LIN {X 0,Y 363.671,Z 845.185,A -85,B 0,C 180,E1 12162.19,E2 12162.19} C_VEL
LIN {X 0,Y 361.588,Z 841.697,A -85,B 0,C 180,E1 12164.164,E2 12164.164} C_VEL
LIN {X 0,Y 357.251,Z 835.619,A -85,B 0,C 180,E1 12167.101,E2 12167.101} C_VEL
LIN {X 0,Y 357.31,Z 834.842,A -85,B 0,C 180,E1 12167.431,E2 12167.431} C_VEL
LIN {X 0,Y 361.071,Z 816.803,A -85,B 0,C 180,E1 12173.615,E2 12173.615} C_VEL
LIN {X 0,Y 366.874,Z 793.95,A -85,B 0,C 180,E1 12179.237,E2 12179.237} C_VEL
LIN {X 0,Y 375.007,Z 763.75,A -85,B 0,C 180,E1 12184.589,E2 12184.589} C_VEL
LIN {X 0,Y 383.635,Z 730.788,A -85,B 0,C 180,E1 12188.762,E2 12188.762} C_VEL
LIN {X 0,Y 391.479,Z 697.041,A -85,B 0,C 180,E1 12191.86,E2 12191.86} C_VEL
LIN {X 0,Y 398.91,Z 656.609,A -85,B 0,C 180,E1 12194.4,E2 12194.4} C_VEL
LIN {X 0,Y 399.383,Z 648.133,A -85,B 0,C 180,E1 12194.901,E2 12194.901} C_VEL
LIN {X 0,Y 385.814,Z 616.735,A -85,B 0,C 180,E1 12198.747,E2 12198.747} C_VEL
LIN {X 0,Y 368.99,Z 587.739,A -85,B 0,C 180,E1 12202.995,E2 12202.995} C_VEL
LIN {X 0,Y 356.259,Z 569.433,A -85,B 0,C 180,E1 12206.425,E2 12206.425} C_VEL
LIN {X 0,Y 353.406,Z 564.379,A -85,B 0,C 180,E1 12207.307,E2 12207.307} C_VEL
LIN {X 0,Y 353.308,Z 563.28,A -85,B 0,C 180,E1 12207.531,E2 12207.531} C_VEL
LIN {X 0,Y 353.587,Z 563.28,A -85,B 0,C 180,E1 12214.74,E2 12214.74} C_VEL
LIN {X 0,Y 353.926,Z 563.28,A -85,B 0,C 180,E1 12222.638,E2 12222.638} C_VEL
LIN {X 0,Y 354.275,Z 563.28,A -85,B 0,C 180,E1 12230.193,E2 12230.193} C_VEL
LIN {X 0,Y 354.927,Z 563.28,A -85,B 0,C 180,E1 12237.566,E2 12237.566} C_VEL
LIN {X 0,Y 354.696,Z 563.28,A -85,B 0,C 180,E1 12244.884,E2 12244.884} C_VEL
LIN {X 0,Y 354.337,Z 563.28,A -85,B 0,C 180,E1 12252.297,E2 12252.297} C_VEL
LIN {X 0,Y 353.84,Z 563.28,A -85,B 0,C 180,E1 12260.247,E2 12260.247} C_VEL
LIN {X 0,Y 353.553,Z 563.28,A -85,B 0,C 180,E1 12268.004,E2 12268.004} C_VEL
LIN {X 0,Y 353.436,Z 563.28,A -85,B 0,C 180,E1 12275.787,E2 12275.787} C_VEL
LIN {X 0,Y 353.192,Z 563.28,A -85,B 0,C 180,E1 12283.423,E2 12283.423} C_VEL
LIN {X 0,Y 353.306,Z 563.28,A -85,B 0,C 180,E1 12290.249,E2 12290.249} C_VEL
LIN {X 0,Y 353.41,Z 564.08,A -85,B 0,C 180,E1 12293.675,E2 12293.675} C_VEL
LIN {X 0,Y 355.308,Z 568.353,A -85,B 0,C 180,E1 12296.796,E2 12296.796} C_VEL
LIN {X 0,Y 359.309,Z 570.875,A -85,B 0,C 180,E1 12303.148,E2 12303.148} C_VEL
LIN {X 0,Y 360.621,Z 572.122,A -85,B 0,C 180,E1 12305.652,E2 12305.652} C_VEL
LIN {X 0,Y 362.642,Z 576.09,A -85,B 0,C 180,E1 12310.557,E2 12310.557} C_VEL
LIN {X 0,Y 364.977,Z 577.856,A -85,B 0,C 180,E1 12317.261,E2 12317.261} C_VEL
LIN {X 0,Y 366.337,Z 578.371,A -85,B 0,C 180,E1 12322.903,E2 12322.903} C_VEL
LIN {X 0,Y 366.937,Z 578.462,A -85,B 0,C 180,E1 12330.001,E2 12330.001} C_VEL
LIN {X 0,Y 366.335,Z 578.387,A -85,B 0,C 180,E1 12337.1,E2 12337.1} C_VEL
LIN {X 0,Y 364.743,Z 577.75,A -85,B 0,C 180,E1 12343.57,E2 12343.57} C_VEL
LIN {X 0,Y 362.374,Z 575.801,A -85,B 0,C 180,E1 12350.065,E2 12350.065} C_VEL
LIN {X 0,Y 360.594,Z 571.886,A -85,B 0,C 180,E1 12354.449,E2 12354.449} C_VEL
LIN {X 0,Y 356.588,Z 569.679,A -85,B 0,C 180,E1 12361.221,E2 12361.221} C_VEL
LIN {X 0,Y 353.659,Z 565.515,A -85,B 0,C 180,E1 12365.832,E2 12365.832} C_VEL
LIN {X 0,Y 353.31,Z 563.28,A -85,B 0,C 180,E1 12366.725,E2 12366.725} C_VEL
LIN {X 0,Y 353.255,Z 563.28,A -85,B 0,C 180,E1 12373.429,E2 12373.429} C_VEL
LIN {X 0,Y 353.304,Z 563.28,A -85,B 0,C 180,E1 12380.248,E2 12380.248} C_VEL
LIN {X 0,Y 353.291,Z 563.28,A -85,B 0,C 180,E1 12386.268,E2 12386.268} C_VEL
LIN {X 0,Y 353.514,Z 563.28,A -85,B 0,C 180,E1 12393.692,E2 12393.692} C_VEL
LIN {X 0,Y 353.865,Z 563.28,A -85,B 0,C 180,E1 12400.051,E2 12400.051} C_VEL
LIN {X 0,Y 354.167,Z 563.28,A -85,B 0,C 180,E1 12407.697,E2 12407.697} C_VEL
LIN {X 0,Y 354.686,Z 563.28,A -85,B 0,C 180,E1 12415.116,E2 12415.116} C_VEL
LIN {X 0,Y 354.947,Z 563.28,A -85,B 0,C 180,E1 12419.997,E2 12419.997} C_VEL
LIN {X 0,Y 354.533,Z 563.28,A -85,B 0,C 180,E1 12427.333,E2 12427.333} C_VEL
LIN {X 0,Y 354.204,Z 563.28,A -85,B 0,C 180,E1 12434.807,E2 12434.807} C_VEL
LIN {X 0,Y 353.755,Z 563.28,A -85,B 0,C 180,E1 12442.573,E2 12442.573} C_VEL
LIN {X 0,Y 353.544,Z 563.28,A -85,B 0,C 180,E1 12447.999,E2 12447.999} C_VEL
LIN {X 0,Y 353.5,Z 563.901,A -85,B 0,C 180,E1 12452.699,E2 12452.699} C_VEL
LIN {X 0,Y 356.151,Z 569.235,A -85,B 0,C 180,E1 12453.542,E2 12453.542} C_VEL
LIN {X 0,Y 358.926,Z 573.181,A -85,B 0,C 180,E1 12454.336,E2 12454.336} C_VEL
LIN {X 0,Y 373.428,Z 594.714,A -85,B 0,C 180,E1 12458.126,E2 12458.126} C_VEL
LIN {X 0,Y 389.979,Z 625.192,A -85,B 0,C 180,E1 12462.337,E2 12462.337} C_VEL
LIN {X 0,Y 399.94,Z 650.173,A -85,B 0,C 180,E1 12465.308,E2 12465.308} C_VEL
LIN {X 0,Y 393.844,Z 685.837,A -85,B 0,C 180,E1 12467.335,E2 12467.335} C_VEL
LIN {X 0,Y 385.413,Z 723.656,A -85,B 0,C 180,E1 12470.49,E2 12470.49} C_VEL
LIN {X 0,Y 377.04,Z 756.232,A -85,B 0,C 180,E1 12474.349,E2 12474.349} C_VEL
LIN {X 0,Y 368.957,Z 786.062,A -85,B 0,C 180,E1 12479.185,E2 12479.185} C_VEL
LIN {X 0,Y 362.194,Z 812.082,A -85,B 0,C 180,E1 12485.048,E2 12485.048} C_VEL
LIN {X 0,Y 358.052,Z 830.361,A -85,B 0,C 180,E1 12490.811,E2 12490.811} C_VEL
LIN {X 0,Y 355.896,Z 844.415,A -85,B 0,C 180,E1 12497.199,E2 12497.199} C_VEL
LIN {X 0,Y 355.194,Z 851.737,A -85,B 0,C 180,E1 12502.676,E2 12502.676} C_VEL
LIN {X 0,Y 355.069,Z 854.938,A -85,B 0,C 180,E1 12507.563,E2 12507.563} C_VEL
LIN {X 0,Y 355.088,Z 854.939,A -85,B 0,C 180,E1 12512.434,E2 12512.434} C_VEL
LIN {X 0,Y 355.305,Z 850.4,A -85,B 0,C 180,E1 12518.547,E2 12518.547} C_VEL
LIN {X 0,Y 356.324,Z 840.794,A -85,B 0,C 180,E1 12524.719,E2 12524.719} C_VEL
LIN {X 0,Y 357.31,Z 834.842,A -85,B 0,C 180,E1 12527.431,E2 12527.431} C_VEL
LIN {X 0,Y 356.685,Z 831.732,A -85,B 0,C 180,E1 12528.738,E2 12528.738} C_VEL
LIN {X 0,Y 352.209,Z 822.528,A -85,B 0,C 180,E1 12532.298,E2 12532.298} C_VEL
LIN {X 0,Y 352.36,Z 821.58,A -85,B 0,C 180,E1 12532.62,E2 12532.62} C_VEL
LIN {X 0,Y 358.152,Z 799.224,A -85,B 0,C 180,E1 12538.636,E2 12538.636} C_VEL
LIN {X 0,Y 365.443,Z 773.594,A -85,B 0,C 180,E1 12543.697,E2 12543.697} C_VEL
LIN {X 0,Y 374.852,Z 740.263,A -85,B 0,C 180,E1 12548.426,E2 12548.426} C_VEL
LIN {X 0,Y 383.311,Z 706.501,A -85,B 0,C 180,E1 12551.853,E2 12551.853} C_VEL
LIN {X 0,Y 391.215,Z 668.882,A -85,B 0,C 180,E1 12554.532,E2 12554.532} C_VEL
LIN {X 0,Y 393.652,Z 652,A -85,B 0,C 180,E1 12555.466,E2 12555.466} C_VEL
LIN {X 0,Y 380.35,Z 620.223,A -85,B 0,C 180,E1 12559.517,E2 12559.517} C_VEL
LIN {X 0,Y 364.483,Z 592.576,A -85,B 0,C 180,E1 12563.775,E2 12563.775} C_VEL
LIN {X 0,Y 351.882,Z 574.587,A -85,B 0,C 180,E1 12567.315,E2 12567.315} C_VEL
LIN {X 0,Y 348.505,Z 569.513,A -85,B 0,C 180,E1 12568.377,E2 12568.377} C_VEL
LIN {X 0,Y 345.524,Z 564.479,A -85,B 0,C 180,E1 12569.381,E2 12569.381} C_VEL
LIN {X 0,Y 345.407,Z 563.28,A -85,B 0,C 180,E1 12569.696,E2 12569.696} C_VEL
LIN {X 0,Y 345.745,Z 563.28,A -85,B 0,C 180,E1 12576.874,E2 12576.874} C_VEL
LIN {X 0,Y 346.098,Z 563.28,A -85,B 0,C 180,E1 12584.838,E2 12584.838} C_VEL
LIN {X 0,Y 346.567,Z 563.28,A -85,B 0,C 180,E1 12592.497,E2 12592.497} C_VEL
LIN {X 0,Y 347.065,Z 563.28,A -85,B 0,C 180,E1 12600.003,E2 12600.003} C_VEL
LIN {X 0,Y 346.585,Z 563.28,A -85,B 0,C 180,E1 12607.508,E2 12607.508} C_VEL
LIN {X 0,Y 346.201,Z 563.28,A -85,B 0,C 180,E1 12615.163,E2 12615.163} C_VEL
LIN {X 0,Y 345.783,Z 563.28,A -85,B 0,C 180,E1 12623.129,E2 12623.129} C_VEL
LIN {X 0,Y 345.532,Z 563.28,A -85,B 0,C 180,E1 12629.142,E2 12629.142} C_VEL
LIN {X 0,Y 345.496,Z 563.28,A -85,B 0,C 180,E1 12634.599,E2 12634.599} C_VEL
LIN {X 0,Y 345.221,Z 563.28,A -85,B 0,C 180,E1 12642.006,E2 12642.006} C_VEL
LIN {X 0,Y 345.236,Z 564.112,A -85,B 0,C 180,E1 12644.299,E2 12644.299} C_VEL
LIN {X 0,Y 347.221,Z 568.468,A -85,B 0,C 180,E1 12647.012,E2 12647.012} C_VEL
LIN {X 0,Y 352.224,Z 571.904,A -85,B 0,C 180,E1 12653.411,E2 12653.411} C_VEL
LIN {X 0,Y 354.534,Z 576.458,A -85,B 0,C 180,E1 12657.128,E2 12657.128} C_VEL
LIN {X 0,Y 358.695,Z 578.802,A -85,B 0,C 180,E1 12663.756,E2 12663.756} C_VEL
LIN {X 0,Y 359.613,Z 580.385,A -85,B 0,C 180,E1 12665.675,E2 12665.675} C_VEL
LIN {X 0,Y 362.06,Z 584.381,A -85,B 0,C 180,E1 12671.471,E2 12671.471} C_VEL
LIN {X 0,Y 364.301,Z 585.783,A -85,B 0,C 180,E1 12678.048,E2 12678.048} C_VEL
LIN {X 0,Y 365.704,Z 586.297,A -85,B 0,C 180,E1 12685.267,E2 12685.267} C_VEL
LIN {X 0,Y 365.909,Z 586.287,A -85,B 0,C 180,E1 12692.365,E2 12692.365} C_VEL
LIN {X 0,Y 364.899,Z 586.104,A -85,B 0,C 180,E1 12699.523,E2 12699.523} C_VEL
LIN {X 0,Y 362.809,Z 584.931,A -85,B 0,C 180,E1 12706.621,E2 12706.621} C_VEL
LIN {X 0,Y 360.101,Z 581.658,A -85,B 0,C 180,E1 12713.228,E2 12713.228} C_VEL
LIN {X 0,Y 359.173,Z 578.883,A -85,B 0,C 180,E1 12715.463,E2 12715.463} C_VEL
LIN {X 0,Y 354.995,Z 577.053,A -85,B 0,C 180,E1 12722.14,E2 12722.14} C_VEL
LIN {X 0,Y 352.286,Z 572.512,A -85,B 0,C 180,E1 12726.42,E2 12726.42} C_VEL
LIN {X 0,Y 351.69,Z 571.028,A -85,B 0,C 180,E1 12727.405,E2 12727.405} C_VEL
LIN {X 0,Y 347.021,Z 568.132,A -85,B 0,C 180,E1 12733.255,E2 12733.255} C_VEL
LIN {X 0,Y 345.297,Z 564.151,A -85,B 0,C 180,E1 12735.632,E2 12735.632} C_VEL
LIN {X 0,Y 345.257,Z 563.28,A -85,B 0,C 180,E1 12737.991,E2 12737.991} C_VEL
LIN {X 0,Y 345.341,Z 563.28,A -85,B 0,C 180,E1 12745.383,E2 12745.383} C_VEL
LIN {X 0,Y 345.466,Z 563.28,A -85,B 0,C 180,E1 12751.28,E2 12751.28} C_VEL
LIN {X 0,Y 345.767,Z 563.28,A -85,B 0,C 180,E1 12756.87,E2 12756.87} C_VEL
LIN {X 0,Y 346.086,Z 563.28,A -85,B 0,C 180,E1 12764.832,E2 12764.832} C_VEL
LIN {X 0,Y 346.582,Z 563.28,A -85,B 0,C 180,E1 12772.492,E2 12772.492} C_VEL
LIN {X 0,Y 347.047,Z 563.28,A -85,B 0,C 180,E1 12777.505,E2 12777.505} C_VEL
LIN {X 0,Y 346.768,Z 563.28,A -85,B 0,C 180,E1 12784.99,E2 12784.99} C_VEL
LIN {X 0,Y 346.396,Z 563.28,A -85,B 0,C 180,E1 12792.578,E2 12792.578} C_VEL
LIN {X 0,Y 345.901,Z 563.28,A -85,B 0,C 180,E1 12800.423,E2 12800.423} C_VEL
LIN {X 0,Y 345.693,Z 563.28,A -85,B 0,C 180,E1 12805.878,E2 12805.878} C_VEL
LIN {X 0,Y 345.599,Z 564.041,A -85,B 0,C 180,E1 12810.622,E2 12810.622} C_VEL
LIN {X 0,Y 348.222,Z 569.222,A -85,B 0,C 180,E1 12811.537,E2 12811.537} C_VEL
LIN {X 0,Y 350.847,Z 572.607,A -85,B 0,C 180,E1 12812.349,E2 12812.349} C_VEL
LIN {X 0,Y 366.964,Z 596.388,A -85,B 0,C 180,E1 12816.899,E2 12816.899} C_VEL
LIN {X 0,Y 383.207,Z 626.372,A -85,B 0,C 180,E1 12821.302,E2 12821.302} C_VEL
LIN {X 0,Y 393.715,Z 651.973,A -85,B 0,C 180,E1 12824.541,E2 12824.541} C_VEL
LIN {X 0,Y 387.168,Z 689.313,A -85,B 0,C 180,E1 12826.802,E2 12826.802} C_VEL
LIN {X 0,Y 378.838,Z 724.988,A -85,B 0,C 180,E1 12829.868,E2 12829.868} C_VEL
LIN {X 0,Y 369.612,Z 759.114,A -85,B 0,C 180,E1 12834.062,E2 12834.062} C_VEL
LIN {X 0,Y 361.647,Z 786.824,A -85,B 0,C 180,E1 12838.727,E2 12838.727} C_VEL
LIN {X 0,Y 355.017,Z 810.994,A -85,B 0,C 180,E1 12844.275,E2 12844.275} C_VEL
LIN {X 0,Y 350.395,Z 830.074,A -85,B 0,C 180,E1 12850.361,E2 12850.361} C_VEL
LIN {X 0,Y 348.045,Z 844.165,A -85,B 0,C 180,E1 12856.906,E2 12856.906} C_VEL
LIN {X 0,Y 347.317,Z 851.491,A -85,B 0,C 180,E1 12862.509,E2 12862.509} C_VEL
LIN {X 0,Y 347.117,Z 854.922,A -85,B 0,C 180,E1 12868.878,E2 12868.878} C_VEL
LIN {X 0,Y 347.209,Z 854.695,A -85,B 0,C 180,E1 12872.49,E2 12872.49} C_VEL
LIN {X 0,Y 347.42,Z 850.153,A -85,B 0,C 180,E1 12878.743,E2 12878.743} C_VEL
LIN {X 0,Y 348.528,Z 840.543,A -85,B 0,C 180,E1 12885.056,E2 12885.056} C_VEL
LIN {X 0,Y 351.495,Z 825.207,A -85,B 0,C 180,E1 12891.401,E2 12891.401} C_VEL
LIN {X 0,Y 352.36,Z 821.58,A -85,B 0,C 180,E1 12892.62,E2 12892.62} C_VEL
LIN {X 0,Y 350.509,Z 813.946,A -85,B 0,C 180,E1 12895.176,E2 12895.176} C_VEL
LIN {X 0,Y 349.082,Z 805.529,A -85,B 0,C 180,E1 12897.691,E2 12897.691} C_VEL
LIN {X 0,Y 356.46,Z 780.665,A -85,B 0,C 180,E1 12903.09,E2 12903.09} C_VEL
LIN {X 0,Y 365.494,Z 750.497,A -85,B 0,C 180,E1 12907.888,E2 12907.888} C_VEL
LIN {X 0,Y 374.925,Z 716.168,A -85,B 0,C 180,E1 12911.766,E2 12911.766} C_VEL
LIN {X 0,Y 382.897,Z 681.994,A -85,B 0,C 180,E1 12914.525,E2 12914.525} C_VEL
LIN {X 0,Y 387.365,Z 654.079,A -85,B 0,C 180,E1 12916.257,E2 12916.257} C_VEL
LIN {X 0,Y 374.283,Z 622.504,A -85,B 0,C 180,E1 12920.489,E2 12920.489} C_VEL
LIN {X 0,Y 358.211,Z 594.506,A -85,B 0,C 180,E1 12925.078,E2 12925.078} C_VEL
LIN {X 0,Y 345.012,Z 575.716,A -85,B 0,C 180,E1 12929.078,E2 12929.078} C_VEL
LIN {X 0,Y 340.974,Z 569.777,A -85,B 0,C 180,E1 12930.466,E2 12930.466} C_VEL
LIN {X 0,Y 337.71,Z 564.923,A -85,B 0,C 180,E1 12931.661,E2 12931.661} C_VEL
LIN {X 0,Y 337.55,Z 563.28,A -85,B 0,C 180,E1 12932.01,E2 12932.01} C_VEL
LIN {X 0,Y 337.978,Z 563.28,A -85,B 0,C 180,E1 12939.651,E2 12939.651} C_VEL
LIN {X 0,Y 338.288,Z 563.28,A -85,B 0,C 180,E1 12947.116,E2 12947.116} C_VEL
LIN {X 0,Y 338.825,Z 563.28,A -85,B 0,C 180,E1 12954.892,E2 12954.892} C_VEL
LIN {X 0,Y 339.163,Z 563.28,A -85,B 0,C 180,E1 12960.003,E2 12960.003} C_VEL
LIN {X 0,Y 338.65,Z 563.28,A -85,B 0,C 180,E1 12967.685,E2 12967.685} C_VEL
LIN {X 0,Y 338.26,Z 563.28,A -85,B 0,C 180,E1 12975.528,E2 12975.528} C_VEL
LIN {X 0,Y 337.94,Z 563.28,A -85,B 0,C 180,E1 12980.932,E2 12980.932} C_VEL
LIN {X 0,Y 337.687,Z 563.28,A -85,B 0,C 180,E1 12986.657,E2 12986.657} C_VEL
LIN {X 0,Y 337.582,Z 563.28,A -85,B 0,C 180,E1 12992.442,E2 12992.442} C_VEL
LIN {X 0,Y 337.414,Z 564.037,A -85,B 0,C 180,E1 12996.425,E2 12996.425} C_VEL
LIN {X 0,Y 339.634,Z 568.903,A -85,B 0,C 180,E1 12999.18,E2 12999.18} C_VEL
LIN {X 0,Y 343.94,Z 571.904,A -85,B 0,C 180,E1 13003.953,E2 13003.953} C_VEL
LIN {X 0,Y 346.648,Z 576.829,A -85,B 0,C 180,E1 13007.56,E2 13007.56} C_VEL
LIN {X 0,Y 351.098,Z 579.793,A -85,B 0,C 180,E1 13013.224,E2 13013.224} C_VEL
LIN {X 0,Y 353.773,Z 584.552,A -85,B 0,C 180,E1 13017.461,E2 13017.461} C_VEL
LIN {X 0,Y 357.821,Z 586.644,A -85,B 0,C 180,E1 13023.906,E2 13023.906} C_VEL
LIN {X 0,Y 358.684,Z 588.701,A -85,B 0,C 180,E1 13025.848,E2 13025.848} C_VEL
LIN {X 0,Y 361.176,Z 592.319,A -85,B 0,C 180,E1 13031.74,E2 13031.74} C_VEL
LIN {X 0,Y 363.326,Z 593.607,A -85,B 0,C 180,E1 13038.016,E2 13038.016} C_VEL
LIN {X 0,Y 364.74,Z 594.137,A -85,B 0,C 180,E1 13045.255,E2 13045.255} C_VEL
LIN {X 0,Y 364.949,Z 594.099,A -85,B 0,C 180,E1 13052.371,E2 13052.371} C_VEL
LIN {X 0,Y 363.929,Z 593.942,A -85,B 0,C 180,E1 13059.548,E2 13059.548} C_VEL
LIN {X 0,Y 361.909,Z 592.826,A -85,B 0,C 180,E1 13066.457,E2 13066.457} C_VEL
LIN {X 0,Y 359.176,Z 589.635,A -85,B 0,C 180,E1 13073.105,E2 13073.105} C_VEL
LIN {X 0,Y 358.173,Z 586.719,A -85,B 0,C 180,E1 13075.539,E2 13075.539} C_VEL
LIN {X 0,Y 354.029,Z 584.918,A -85,B 0,C 180,E1 13082.137,E2 13082.137} C_VEL
LIN {X 0,Y 351.143,Z 580.278,A -85,B 0,C 180,E1 13086.644,E2 13086.644} C_VEL
LIN {X 0,Y 350.271,Z 578.746,A -85,B 0,C 180,E1 13087.99,E2 13087.99} C_VEL
LIN {X 0,Y 345.694,Z 575.627,A -85,B 0,C 180,E1 13093.655,E2 13093.655} C_VEL
LIN {X 0,Y 343.38,Z 570.929,A -85,B 0,C 180,E1 13096.755,E2 13096.755} C_VEL
LIN {X 0,Y 338.699,Z 567.666,A -85,B 0,C 180,E1 13101.883,E2 13101.883} C_VEL
LIN {X 0,Y 337.303,Z 563.589,A -85,B 0,C 180,E1 13103.736,E2 13103.736} C_VEL
LIN {X 0,Y 337.518,Z 563.28,A -85,B 0,C 180,E1 13110.539,E2 13110.539} C_VEL
LIN {X 0,Y 337.832,Z 563.28,A -85,B 0,C 180,E1 13116.294,E2 13116.294} C_VEL
LIN {X 0,Y 338.024,Z 563.28,A -85,B 0,C 180,E1 13121.788,E2 13121.788} C_VEL
LIN {X 0,Y 338.409,Z 563.28,A -85,B 0,C 180,E1 13129.723,E2 13129.723} C_VEL
LIN {X 0,Y 339.128,Z 563.28,A -85,B 0,C 180,E1 13137.447,E2 13137.447} C_VEL
LIN {X 0,Y 338.842,Z 563.28,A -85,B 0,C 180,E1 13145.107,E2 13145.107} C_VEL
LIN {X 0,Y 338.468,Z 563.28,A -85,B 0,C 180,E1 13152.877,E2 13152.877} C_VEL
LIN {X 0,Y 337.924,Z 563.28,A -85,B 0,C 180,E1 13160.928,E2 13160.928} C_VEL
LIN {X 0,Y 337.632,Z 563.573,A -85,B 0,C 180,E1 13168.256,E2 13168.256} C_VEL
LIN {X 0,Y 339.813,Z 568.738,A -85,B 0,C 180,E1 13169.146,E2 13169.146} C_VEL
LIN {X 0,Y 342.794,Z 572.041,A -85,B 0,C 180,E1 13170.154,E2 13170.154} C_VEL
LIN {X 0,Y 359.439,Z 596.205,A -85,B 0,C 180,E1 13175.279,E2 13175.279} C_VEL
LIN {X 0,Y 376.137,Z 626.656,A -85,B 0,C 180,E1 13180.099,E2 13180.099} C_VEL
LIN {X 0,Y 387.721,Z 655.219,A -85,B 0,C 180,E1 13183.885,E2 13183.885} C_VEL
LIN {X 0,Y 380.122,Z 694.653,A -85,B 0,C 180,E1 13186.388,E2 13186.388} C_VEL
LIN {X 0,Y 371.641,Z 728.551,A -85,B 0,C 180,E1 13189.482,E2 13189.482} C_VEL
LIN {X 0,Y 362.163,Z 761.995,A -85,B 0,C 180,E1 13193.76,E2 13193.76} C_VEL
LIN {X 0,Y 353.372,Z 790.825,A -85,B 0,C 180,E1 13198.916,E2 13198.916} C_VEL
LIN {X 0,Y 346.823,Z 813.809,A -85,B 0,C 180,E1 13204.553,E2 13204.553} C_VEL
LIN {X 0,Y 342.012,Z 833.157,A -85,B 0,C 180,E1 13211.226,E2 13211.226} C_VEL
LIN {X 0,Y 340.079,Z 845.195,A -85,B 0,C 180,E1 13217.456,E2 13217.456} C_VEL
LIN {X 0,Y 339.298,Z 852.286,A -85,B 0,C 180,E1 13223.615,E2 13223.615} C_VEL
LIN {X 0,Y 339.347,Z 854.854,A -85,B 0,C 180,E1 13229.999,E2 13229.999} C_VEL
LIN {X 0,Y 339.254,Z 853.243,A -85,B 0,C 180,E1 13235.103,E2 13235.103} C_VEL
LIN {X 0,Y 339.811,Z 846.898,A -85,B 0,C 180,E1 13241.387,E2 13241.387} C_VEL
LIN {X 0,Y 341.78,Z 834.894,A -85,B 0,C 180,E1 13248.001,E2 13248.001} C_VEL
LIN {X 0,Y 345.864,Z 817.46,A -85,B 0,C 180,E1 13254.348,E2 13254.348} C_VEL
LIN {X 0,Y 349.082,Z 805.529,A -85,B 0,C 180,E1 13257.691,E2 13257.691} C_VEL
LIN {X 0,Y 348.158,Z 796.543,A -85,B 0,C 180,E1 13260.162,E2 13260.162} C_VEL
LIN {X 0,Y 347.612,Z 786.819,A -85,B 0,C 180,E1 13262.567,E2 13262.567} C_VEL
LIN {X 0,Y 356.551,Z 758.624,A -85,B 0,C 180,E1 13267.471,E2 13267.471} C_VEL
LIN {X 0,Y 366.415,Z 725.473,A -85,B 0,C 180,E1 13271.648,E2 13271.648} C_VEL
LIN {X 0,Y 375.662,Z 688.407,A -85,B 0,C 180,E1 13274.914,E2 13274.914} C_VEL
LIN {X 0,Y 381.562,Z 657.868,A -85,B 0,C 180,E1 13276.843,E2 13276.843} C_VEL
LIN {X 0,Y 368.955,Z 626.366,A -85,B 0,C 180,E1 13281.241,E2 13281.241} C_VEL
LIN {X 0,Y 353.883,Z 599.562,A -85,B 0,C 180,E1 13285.859,E2 13285.859} C_VEL
LIN {X 0,Y 338.477,Z 576.893,A -85,B 0,C 180,E1 13290.911,E2 13290.911} C_VEL
LIN {X 0,Y 333.198,Z 569.859,A -85,B 0,C 180,E1 13292.892,E2 13292.892} C_VEL
LIN {X 0,Y 329.909,Z 564.995,A -85,B 0,C 180,E1 13294.255,E2 13294.255} C_VEL
LIN {X 0,Y 329.721,Z 563.28,A -85,B 0,C 180,E1 13294.601,E2 13294.601} C_VEL
LIN {X 0,Y 330.058,Z 563.28,A -85,B 0,C 180,E1 13301.338,E2 13301.338} C_VEL
LIN {X 0,Y 330.487,Z 563.28,A -85,B 0,C 180,E1 13309.479,E2 13309.479} C_VEL
LIN {X 0,Y 331.192,Z 563.28,A -85,B 0,C 180,E1 13317.391,E2 13317.391} C_VEL
LIN {X 0,Y 331.128,Z 563.28,A -85,B 0,C 180,E1 13322.615,E2 13322.615} C_VEL
LIN {X 0,Y 330.585,Z 563.28,A -85,B 0,C 180,E1 13330.523,E2 13330.523} C_VEL
LIN {X 0,Y 330.139,Z 563.28,A -85,B 0,C 180,E1 13338.663,E2 13338.663} C_VEL
LIN {X 0,Y 329.844,Z 563.28,A -85,B 0,C 180,E1 13344.317,E2 13344.317} C_VEL
LIN {X 0,Y 329.741,Z 563.921,A -85,B 0,C 180,E1 13349.428,E2 13349.428} C_VEL
LIN {X 0,Y 331.188,Z 567.963,A -85,B 0,C 180,E1 13351.118,E2 13351.118} C_VEL
LIN {X 0,Y 336.08,Z 571.903,A -85,B 0,C 180,E1 13356.081,E2 13356.081} C_VEL
LIN {X 0,Y 339.131,Z 577.222,A -85,B 0,C 180,E1 13359.702,E2 13359.702} C_VEL
LIN {X 0,Y 342.728,Z 579.756,A -85,B 0,C 180,E1 13363.696,E2 13363.696} C_VEL
LIN {X 0,Y 345.917,Z 584.941,A -85,B 0,C 180,E1 13367.871,E2 13367.871} C_VEL
LIN {X 0,Y 349.963,Z 587.64,A -85,B 0,C 180,E1 13373.013,E2 13373.013} C_VEL
LIN {X 0,Y 352.937,Z 592.55,A -85,B 0,C 180,E1 13377.667,E2 13377.667} C_VEL
LIN {X 0,Y 356.873,Z 594.489,A -85,B 0,C 180,E1 13383.942,E2 13383.942} C_VEL
LIN {X 0,Y 359.25,Z 599.08,A -85,B 0,C 180,E1 13389.33,E2 13389.33} C_VEL
LIN {X 0,Y 361.583,Z 601.103,A -85,B 0,C 180,E1 13395.5,E2 13395.5} C_VEL
LIN {X 0,Y 362.967,Z 601.698,A -85,B 0,C 180,E1 13400.429,E2 13400.429} C_VEL
LIN {X 0,Y 363.979,Z 602.001,A -85,B 0,C 180,E1 13407.625,E2 13407.625} C_VEL
LIN {X 0,Y 363.777,Z 601.961,A -85,B 0,C 180,E1 13414.76,E2 13414.76} C_VEL
LIN {X 0,Y 362.345,Z 601.471,A -85,B 0,C 180,E1 13422.02,E2 13422.02} C_VEL
LIN {X 0,Y 360.067,Z 599.989,A -85,B 0,C 180,E1 13428.754,E2 13428.754} C_VEL
LIN {X 0,Y 357.467,Z 595.699,A -85,B 0,C 180,E1 13434.797,E2 13434.797} C_VEL
LIN {X 0,Y 356.218,Z 594.331,A -85,B 0,C 180,E1 13437.173,E2 13437.173} C_VEL
LIN {X 0,Y 352.058,Z 591.704,A -85,B 0,C 180,E1 13443.697,E2 13443.697} C_VEL
LIN {X 0,Y 349.743,Z 586.894,A -85,B 0,C 180,E1 13447.393,E2 13447.393} C_VEL
LIN {X 0,Y 344.721,Z 583.586,A -85,B 0,C 180,E1 13453.639,E2 13453.639} C_VEL
LIN {X 0,Y 342.364,Z 578.741,A -85,B 0,C 180,E1 13456.807,E2 13456.807} C_VEL
LIN {X 0,Y 337.545,Z 575.41,A -85,B 0,C 180,E1 13462.067,E2 13462.067} C_VEL
LIN {X 0,Y 335.829,Z 571.039,A -85,B 0,C 180,E1 13464.255,E2 13464.255} C_VEL
LIN {X 0,Y 331.03,Z 567.877,A -85,B 0,C 180,E1 13469.032,E2 13469.032} C_VEL
LIN {X 0,Y 329.64,Z 563.879,A -85,B 0,C 180,E1 13470.65,E2 13470.65} C_VEL
LIN {X 0,Y 329.953,Z 563.28,A -85,B 0,C 180,E1 13478.536,E2 13478.536} C_VEL
LIN {X 0,Y 330.323,Z 563.28,A -85,B 0,C 180,E1 13486.794,E2 13486.794} C_VEL
LIN {X 0,Y 330.922,Z 563.28,A -85,B 0,C 180,E1 13494.765,E2 13494.765} C_VEL
LIN {X 0,Y 331.237,Z 563.28,A -85,B 0,C 180,E1 13499.997,E2 13499.997} C_VEL
LIN {X 0,Y 330.732,Z 563.28,A -85,B 0,C 180,E1 13507.864,E2 13507.864} C_VEL
LIN {X 0,Y 330.308,Z 563.28,A -85,B 0,C 180,E1 13515.906,E2 13515.906} C_VEL
LIN {X 0,Y 329.831,Z 563.28,A -85,B 0,C 180,E1 13524.312,E2 13524.312} C_VEL
LIN {X 0,Y 329.753,Z 563.28,A -85,B 0,C 180,E1 13525.583,E2 13525.583} C_VEL
LIN {X 0,Y 331.649,Z 568.354,A -85,B 0,C 180,E1 13526.514,E2 13526.514} C_VEL
LIN {X 0,Y 335.135,Z 572.196,A -85,B 0,C 180,E1 13527.846,E2 13527.846} C_VEL
LIN {X 0,Y 348.91,Z 591.676,A -85,B 0,C 180,E1 13532.577,E2 13532.577} C_VEL
LIN {X 0,Y 363.161,Z 615.427,A -85,B 0,C 180,E1 13536.984,E2 13536.984} C_VEL
LIN {X 0,Y 376.647,Z 644.281,A -85,B 0,C 180,E1 13541.335,E2 13541.335} C_VEL
LIN {X 0,Y 381.733,Z 658.528,A -85,B 0,C 180,E1 13543.238,E2 13543.238} C_VEL
LIN {X 0,Y 373.746,Z 697.132,A -85,B 0,C 180,E1 13545.746,E2 13545.746} C_VEL
LIN {X 0,Y 364.397,Z 732.195,A -85,B 0,C 180,E1 13549.093,E2 13549.093} C_VEL
LIN {X 0,Y 355.331,Z 762.729,A -85,B 0,C 180,E1 13553.139,E2 13553.139} C_VEL
LIN {X 0,Y 346.061,Z 791.659,A -85,B 0,C 180,E1 13558.447,E2 13558.447} C_VEL
LIN {X 0,Y 339.141,Z 814.626,A -85,B 0,C 180,E1 13564.288,E2 13564.288} C_VEL
LIN {X 0,Y 334.271,Z 833.191,A -85,B 0,C 180,E1 13570.894,E2 13570.894} C_VEL
LIN {X 0,Y 332.178,Z 845.347,A -85,B 0,C 180,E1 13577.434,E2 13577.434} C_VEL
LIN {X 0,Y 331.421,Z 852.04,A -85,B 0,C 180,E1 13583.463,E2 13583.463} C_VEL
LIN {X 0,Y 331.46,Z 854.609,A -85,B 0,C 180,E1 13589.999,E2 13589.999} C_VEL
LIN {X 0,Y 331.383,Z 852.041,A -85,B 0,C 180,E1 13596.536,E2 13596.536} C_VEL
LIN {X 0,Y 332.265,Z 844.545,A -85,B 0,C 180,E1 13603.124,E2 13603.124} C_VEL
LIN {X 0,Y 334.73,Z 831.569,A -85,B 0,C 180,E1 13609.759,E2 13609.759} C_VEL
LIN {X 0,Y 339.744,Z 812.489,A -85,B 0,C 180,E1 13616.368,E2 13616.368} C_VEL
LIN {X 0,Y 347.424,Z 787.397,A -85,B 0,C 180,E1 13622.446,E2 13622.446} C_VEL
LIN {X 0,Y 347.612,Z 786.819,A -85,B 0,C 180,E1 13622.567,E2 13622.567} C_VEL
LIN {X 0,Y 347.5,Z 776.544,A -85,B 0,C 180,E1 13624.909,E2 13624.909} C_VEL
LIN {X 0,Y 347.789,Z 765.564,A -85,B 0,C 180,E1 13627.155,E2 13627.155} C_VEL
LIN {X 0,Y 357.563,Z 734.561,A -85,B 0,C 180,E1 13631.455,E2 13631.455} C_VEL
LIN {X 0,Y 367.487,Z 698.723,A -85,B 0,C 180,E1 13634.987,E2 13634.987} C_VEL
LIN {X 0,Y 375.599,Z 660.92,A -85,B 0,C 180,E1 13637.539,E2 13637.539} C_VEL
LIN {X 0,Y 363.254,Z 629.59,A -85,B 0,C 180,E1 13642.14,E2 13642.14} C_VEL
LIN {X 0,Y 348.592,Z 602.601,A -85,B 0,C 180,E1 13647.009,E2 13647.009} C_VEL
LIN {X 0,Y 334.877,Z 582.819,A -85,B 0,C 180,E1 13651.765,E2 13651.765} C_VEL
LIN {X 0,Y 330.133,Z 576.371,A -85,B 0,C 180,E1 13653.629,E2 13653.629} C_VEL
LIN {X 0,Y 326.103,Z 570.274,A -85,B 0,C 180,E1 13655.392,E2 13655.392} C_VEL
LIN {X 0,Y 322.21,Z 565.269,A -85,B 0,C 180,E1 13657.211,E2 13657.211} C_VEL
LIN {X 0,Y 321.969,Z 563.28,A -85,B 0,C 180,E1 13657.696,E2 13657.696} C_VEL
LIN {X 0,Y 322.235,Z 563.28,A -85,B 0,C 180,E1 13663.685,E2 13663.685} C_VEL
LIN {X 0,Y 322.747,Z 563.28,A -85,B 0,C 180,E1 13671.94,E2 13671.94} C_VEL
LIN {X 0,Y 323.271,Z 563.28,A -85,B 0,C 180,E1 13677.327,E2 13677.327} C_VEL
LIN {X 0,Y 323.211,Z 563.28,A -85,B 0,C 180,E1 13682.679,E2 13682.679} C_VEL
LIN {X 0,Y 322.65,Z 563.28,A -85,B 0,C 180,E1 13690.847,E2 13690.847} C_VEL
LIN {X 0,Y 322.337,Z 563.28,A -85,B 0,C 180,E1 13696.316,E2 13696.316} C_VEL
LIN {X 0,Y 322.038,Z 563.667,A -85,B 0,C 180,E1 13703.973,E2 13703.973} C_VEL
LIN {X 0,Y 323.67,Z 568.384,A -85,B 0,C 180,E1 13705.407,E2 13705.407} C_VEL
LIN {X 0,Y 328.207,Z 571.991,A -85,B 0,C 180,E1 13709.058,E2 13709.058} C_VEL
LIN {X 0,Y 331.249,Z 576.956,A -85,B 0,C 180,E1 13712.123,E2 13712.123} C_VEL
LIN {X 0,Y 334.857,Z 579.898,A -85,B 0,C 180,E1 13715.865,E2 13715.865} C_VEL
LIN {X 0,Y 338.432,Z 585.297,A -85,B 0,C 180,E1 13719.995,E2 13719.995} C_VEL
LIN {X 0,Y 341.539,Z 587.571,A -85,B 0,C 180,E1 13723.471,E2 13723.471} C_VEL
LIN {X 0,Y 345.072,Z 592.881,A -85,B 0,C 180,E1 13728.026,E2 13728.026} C_VEL
LIN {X 0,Y 348.838,Z 595.42,A -85,B 0,C 180,E1 13732.801,E2 13732.801} C_VEL
LIN {X 0,Y 351.974,Z 600.412,A -85,B 0,C 180,E1 13737.683,E2 13737.683} C_VEL
LIN {X 0,Y 356.292,Z 603.018,A -85,B 0,C 180,E1 13744.696,E2 13744.696} C_VEL
LIN {X 0,Y 358.582,Z 607.286,A -85,B 0,C 180,E1 13750.118,E2 13750.118} C_VEL
LIN {X 0,Y 360.929,Z 609.081,A -85,B 0,C 180,E1 13756.574,E2 13756.574} C_VEL
LIN {X 0,Y 362.475,Z 609.702,A -85,B 0,C 180,E1 13762.827,E2 13762.827} C_VEL
LIN {X 0,Y 363.089,Z 609.804,A -85,B 0,C 180,E1 13770.001,E2 13770.001} C_VEL
LIN {X 0,Y 362.469,Z 609.744,A -85,B 0,C 180,E1 13777.176,E2 13777.176} C_VEL
LIN {X 0,Y 360.814,Z 609.034,A -85,B 0,C 180,E1 13783.923,E2 13783.923} C_VEL
LIN {X 0,Y 358.266,Z 606.892,A -85,B 0,C 180,E1 13790.73,E2 13790.73} C_VEL
LIN {X 0,Y 355.931,Z 602.346,A -85,B 0,C 180,E1 13796.011,E2 13796.011} C_VEL
LIN {X 0,Y 351.705,Z 600.281,A -85,B 0,C 180,E1 13802.701,E2 13802.701} C_VEL
LIN {X 0,Y 348.776,Z 595.406,A -85,B 0,C 180,E1 13807.282,E2 13807.282} C_VEL
LIN {X 0,Y 343.444,Z 591.115,A -85,B 0,C 180,E1 13814.003,E2 13814.003} C_VEL
LIN {X 0,Y 341.015,Z 586.484,A -85,B 0,C 180,E1 13817.204,E2 13817.204} C_VEL
LIN {X 0,Y 336.294,Z 583.01,A -85,B 0,C 180,E1 13822.366,E2 13822.366} C_VEL
LIN {X 0,Y 333.983,Z 578.67,A -85,B 0,C 180,E1 13825.119,E2 13825.119} C_VEL
LIN {X 0,Y 329.242,Z 574.66,A -85,B 0,C 180,E1 13829.871,E2 13829.871} C_VEL
LIN {X 0,Y 327.44,Z 570.882,A -85,B 0,C 180,E1 13831.654,E2 13831.654} C_VEL
LIN {X 0,Y 322.948,Z 567.333,A -85,B 0,C 180,E1 13835.129,E2 13835.129} C_VEL
LIN {X 0,Y 322.039,Z 563.28,A -85,B 0,C 180,E1 13836.256,E2 13836.256} C_VEL
LIN {X 0,Y 322.239,Z 563.28,A -85,B 0,C 180,E1 13843.679,E2 13843.679} C_VEL
LIN {X 0,Y 322.761,Z 563.28,A -85,B 0,C 180,E1 13851.934,E2 13851.934} C_VEL
LIN {X 0,Y 323.287,Z 563.28,A -85,B 0,C 180,E1 13857.322,E2 13857.322} C_VEL
LIN {X 0,Y 323.179,Z 563.28,A -85,B 0,C 180,E1 13862.673,E2 13862.673} C_VEL
LIN {X 0,Y 322.665,Z 563.28,A -85,B 0,C 180,E1 13870.848,E2 13870.848} C_VEL
LIN {X 0,Y 322.35,Z 563.28,A -85,B 0,C 180,E1 13876.309,E2 13876.309} C_VEL
LIN {X 0,Y 321.99,Z 563.385,A -85,B 0,C 180,E1 13882.591,E2 13882.591} C_VEL
LIN {X 0,Y 323.8,Z 568.301,A -85,B 0,C 180,E1 13883.606,E2 13883.606} C_VEL
LIN {X 0,Y 327.325,Z 571.877,A -85,B 0,C 180,E1 13885.147,E2 13885.147} C_VEL
LIN {X 0,Y 333.711,Z 581.227,A -85,B 0,C 180,E1 13887.792,E2 13887.792} C_VEL
LIN {X 0,Y 343.182,Z 594.556,A -85,B 0,C 180,E1 13891.203,E2 13891.203} C_VEL
LIN {X 0,Y 357.42,Z 617.945,A -85,B 0,C 180,E1 13895.901,E2 13895.901} C_VEL
LIN {X 0,Y 370.95,Z 647.719,A -85,B 0,C 180,E1 13900.604,E2 13900.604} C_VEL
LIN {X 0,Y 375.597,Z 662.076,A -85,B 0,C 180,E1 13902.559,E2 13902.559} C_VEL
LIN {X 0,Y 367.564,Z 698.728,A -85,B 0,C 180,E1 13905.025,E2 13905.025} C_VEL
LIN {X 0,Y 357.593,Z 734.543,A -85,B 0,C 180,E1 13908.546,E2 13908.546} C_VEL
LIN {X 0,Y 347.628,Z 766.008,A -85,B 0,C 180,E1 13912.918,E2 13912.918} C_VEL
LIN {X 0,Y 338.183,Z 794.381,A -85,B 0,C 180,E1 13918.378,E2 13918.378} C_VEL
LIN {X 0,Y 330.481,Z 818.657,A -85,B 0,C 180,E1 13925.015,E2 13925.015} C_VEL
LIN {X 0,Y 326.262,Z 834.381,A -85,B 0,C 180,E1 13931.108,E2 13931.108} C_VEL
LIN {X 0,Y 324.217,Z 846.015,A -85,B 0,C 180,E1 13937.78,E2 13937.78} C_VEL
LIN {X 0,Y 323.479,Z 852.75,A -85,B 0,C 180,E1 13944.645,E2 13944.645} C_VEL
LIN {X 0,Y 323.561,Z 854.364,A -85,B 0,C 180,E1 13949.999,E2 13949.999} C_VEL
LIN {X 0,Y 323.511,Z 851.795,A -85,B 0,C 180,E1 13956.695,E2 13956.695} C_VEL
LIN {X 0,Y 324.459,Z 844.296,A -85,B 0,C 180,E1 13963.446,E2 13963.446} C_VEL
LIN {X 0,Y 327.066,Z 831.312,A -85,B 0,C 180,E1 13970.244,E2 13970.244} C_VEL
LIN {X 0,Y 332.425,Z 812.234,A -85,B 0,C 180,E1 13976.995,E2 13976.995} C_VEL
LIN {X 0,Y 340.444,Z 787.461,A -85,B 0,C 180,E1 13983.116,E2 13983.116} C_VEL
LIN {X 0,Y 347.789,Z 765.564,A -85,B 0,C 180,E1 13987.155,E2 13987.155} C_VEL
LIN {X 0,Y 348.437,Z 754.02,A -85,B 0,C 180,E1 13989.321,E2 13989.321} C_VEL
LIN {X 0,Y 349.154,Z 741.862,A -85,B 0,C 180,E1 13991.391,E2 13991.391} C_VEL
LIN {X 0,Y 359.251,Z 708.28,A -85,B 0,C 180,E1 13995.029,E2 13995.029} C_VEL
LIN {X 0,Y 368.775,Z 669.481,A -85,B 0,C 180,E1 13997.915,E2 13997.915} C_VEL
LIN {X 0,Y 369.36,Z 663.289,A -85,B 0,C 180,E1 13998.374,E2 13998.374} C_VEL
LIN {X 0,Y 357.97,Z 633.456,A -85,B 0,C 180,E1 14002.956,E2 14002.956} C_VEL
LIN {X 0,Y 344.724,Z 608.406,A -85,B 0,C 180,E1 14007.681,E2 14007.681} C_VEL
LIN {X 0,Y 331.226,Z 588.249,A -85,B 0,C 180,E1 14012.702,E2 14012.702} C_VEL
LIN {X 0,Y 323.205,Z 576.993,A -85,B 0,C 180,E1 14016.166,E2 14016.166} C_VEL
LIN {X 0,Y 319.553,Z 571.213,A -85,B 0,C 180,E1 14018.012,E2 14018.012} C_VEL
LIN {X 0,Y 314.646,Z 565.98,A -85,B 0,C 180,E1 14020.661,E2 14020.661} C_VEL
LIN {X 0,Y 314.171,Z 563.28,A -85,B 0,C 180,E1 14021.267,E2 14021.267} C_VEL
LIN {X 0,Y 314.591,Z 563.28,A -85,B 0,C 180,E1 14028.941,E2 14028.941} C_VEL
LIN {X 0,Y 315.365,Z 563.28,A -85,B 0,C 180,E1 14037.26,E2 14037.26} C_VEL
LIN {X 0,Y 315.316,Z 563.28,A -85,B 0,C 180,E1 14042.746,E2 14042.746} C_VEL
LIN {X 0,Y 314.741,Z 563.28,A -85,B 0,C 180,E1 14051.059,E2 14051.059} C_VEL
LIN {X 0,Y 314.261,Z 563.28,A -85,B 0,C 180,E1 14059.279,E2 14059.279} C_VEL
LIN {X 0,Y 316.144,Z 568.549,A -85,B 0,C 180,E1 14060.836,E2 14060.836} C_VEL
LIN {X 0,Y 320.382,Z 572.141,A -85,B 0,C 180,E1 14063.605,E2 14063.605} C_VEL
LIN {X 0,Y 323.431,Z 577.104,A -85,B 0,C 180,E1 14066.026,E2 14066.026} C_VEL
LIN {X 0,Y 326.782,Z 579.712,A -85,B 0,C 180,E1 14068.725,E2 14068.725} C_VEL
LIN {X 0,Y 330.263,Z 584.891,A -85,B 0,C 180,E1 14072.131,E2 14072.131} C_VEL
LIN {X 0,Y 333.641,Z 587.665,A -85,B 0,C 180,E1 14075.625,E2 14075.625} C_VEL
LIN {X 0,Y 337.232,Z 593.016,A -85,B 0,C 180,E1 14079.773,E2 14079.773} C_VEL
LIN {X 0,Y 340.321,Z 595.292,A -85,B 0,C 180,E1 14083.198,E2 14083.198} C_VEL
LIN {X 0,Y 344.094,Z 600.763,A -85,B 0,C 180,E1 14088.027,E2 14088.027} C_VEL
LIN {X 0,Y 347.758,Z 603.344,A -85,B 0,C 180,E1 14092.666,E2 14092.666} C_VEL
LIN {X 0,Y 351.141,Z 608.406,A -85,B 0,C 180,E1 14097.886,E2 14097.886} C_VEL
LIN {X 0,Y 355.301,Z 611.12,A -85,B 0,C 180,E1 14104.703,E2 14104.703} C_VEL
LIN {X 0,Y 357.961,Z 615.546,A -85,B 0,C 180,E1 14110.898,E2 14110.898} C_VEL
LIN {X 0,Y 360.4,Z 617.081,A -85,B 0,C 180,E1 14117.917,E2 14117.917} C_VEL
LIN {X 0,Y 361.847,Z 617.656,A -85,B 0,C 180,E1 14125.217,E2 14125.217} C_VEL
LIN {X 0,Y 362.06,Z 617.621,A -85,B 0,C 180,E1 14132.39,E2 14132.39} C_VEL
LIN {X 0,Y 361.013,Z 617.456,A -85,B 0,C 180,E1 14139.626,E2 14139.626} C_VEL
LIN {X 0,Y 358.954,Z 616.294,A -85,B 0,C 180,E1 14146.605,E2 14146.605} C_VEL
LIN {X 0,Y 356.14,Z 613.076,A -85,B 0,C 180,E1 14153.393,E2 14153.393} C_VEL
LIN {X 0,Y 354.581,Z 610.067,A -85,B 0,C 180,E1 14156.653,E2 14156.653} C_VEL
LIN {X 0,Y 350.386,Z 607.759,A -85,B 0,C 180,E1 14163.273,E2 14163.273} C_VEL
LIN {X 0,Y 347.508,Z 602.686,A -85,B 0,C 180,E1 14167.753,E2 14167.753} C_VEL
LIN {X 0,Y 342.321,Z 598.873,A -85,B 0,C 180,E1 14174.179,E2 14174.179} C_VEL
LIN {X 0,Y 339.51,Z 594.153,A -85,B 0,C 180,E1 14177.775,E2 14177.775} C_VEL
LIN {X 0,Y 334.926,Z 590.382,A -85,B 0,C 180,E1 14182.827,E2 14182.827} C_VEL
LIN {X 0,Y 332.867,Z 586.464,A -85,B 0,C 180,E1 14185.257,E2 14185.257} C_VEL
LIN {X 0,Y 327.963,Z 582.312,A -85,B 0,C 180,E1 14190.139,E2 14190.139} C_VEL
LIN {X 0,Y 325.9,Z 578.531,A -85,B 0,C 180,E1 14192.113,E2 14192.113} C_VEL
LIN {X 0,Y 321.277,Z 574.607,A -85,B 0,C 180,E1 14195.588,E2 14195.588} C_VEL
LIN {X 0,Y 319.364,Z 570.73,A -85,B 0,C 180,E1 14197.109,E2 14197.109} C_VEL
LIN {X 0,Y 314.984,Z 566.828,A -85,B 0,C 180,E1 14199.918,E2 14199.918} C_VEL
LIN {X 0,Y 314.189,Z 563.28,A -85,B 0,C 180,E1 14200.716,E2 14200.716} C_VEL
LIN {X 0,Y 314.606,Z 563.28,A -85,B 0,C 180,E1 14208.936,E2 14208.936} C_VEL
LIN {X 0,Y 315.381,Z 563.28,A -85,B 0,C 180,E1 14217.255,E2 14217.255} C_VEL
LIN {X 0,Y 315.291,Z 563.28,A -85,B 0,C 180,E1 14222.74,E2 14222.74} C_VEL
LIN {X 0,Y 314.757,Z 563.28,A -85,B 0,C 180,E1 14231.053,E2 14231.053} C_VEL
LIN {X 0,Y 314.273,Z 563.803,A -85,B 0,C 180,E1 14238.999,E2 14238.999} C_VEL
LIN {X 0,Y 316.389,Z 568.807,A -85,B 0,C 180,E1 14240.388,E2 14240.388} C_VEL
LIN {X 0,Y 319.702,Z 571.671,A -85,B 0,C 180,E1 14242.081,E2 14242.081} C_VEL
LIN {X 0,Y 324.099,Z 577.654,A -85,B 0,C 180,E1 14244.221,E2 14244.221} C_VEL
LIN {X 0,Y 338.892,Z 599.046,A -85,B 0,C 180,E1 14250.223,E2 14250.223} C_VEL
LIN {X 0,Y 353.328,Z 623.778,A -85,B 0,C 180,E1 14255.355,E2 14255.355} C_VEL
LIN {X 0,Y 365.964,Z 652.937,A -85,B 0,C 180,E1 14260.108,E2 14260.108} C_VEL
LIN {X 0,Y 369.596,Z 665.144,A -85,B 0,C 180,E1 14261.829,E2 14261.829} C_VEL
LIN {X 0,Y 361.031,Z 701.709,A -85,B 0,C 180,E1 14264.403,E2 14264.403} C_VEL
LIN {X 0,Y 350.807,Z 736.889,A -85,B 0,C 180,E1 14267.976,E2 14267.976} C_VEL
LIN {X 0,Y 339.96,Z 769.225,A -85,B 0,C 180,E1 14272.677,E2 14272.677} C_VEL
LIN {X 0,Y 330.547,Z 795.987,A -85,B 0,C 180,E1 14278.089,E2 14278.089} C_VEL
LIN {X 0,Y 322.773,Z 819.463,A -85,B 0,C 180,E1 14284.746,E2 14284.746} C_VEL
LIN {X 0,Y 318.21,Z 835.88,A -85,B 0,C 180,E1 14291.508,E2 14291.508} C_VEL
LIN {X 0,Y 316.355,Z 845.765,A -85,B 0,C 180,E1 14297.471,E2 14297.471} C_VEL
LIN {X 0,Y 315.596,Z 852.504,A -85,B 0,C 180,E1 14304.511,E2 14304.511} C_VEL
LIN {X 0,Y 315.672,Z 854.119,A -85,B 0,C 180,E1 14309.999,E2 14309.999} C_VEL
LIN {X 0,Y 315.623,Z 851.548,A -85,B 0,C 180,E1 14316.863,E2 14316.863} C_VEL
LIN {X 0,Y 316.617,Z 844.046,A -85,B 0,C 180,E1 14323.785,E2 14323.785} C_VEL
LIN {X 0,Y 319.441,Z 831.059,A -85,B 0,C 180,E1 14330.749,E2 14330.749} C_VEL
LIN {X 0,Y 325.171,Z 811.981,A -85,B 0,C 180,E1 14337.648,E2 14337.648} C_VEL
LIN {X 0,Y 333.829,Z 786.616,A -85,B 0,C 180,E1 14344.012,E2 14344.012} C_VEL
LIN {X 0,Y 343.565,Z 758.753,A -85,B 0,C 180,E1 14349.027,E2 14349.027} C_VEL
LIN {X 0,Y 349.154,Z 741.862,A -85,B 0,C 180,E1 14351.391,E2 14351.391} C_VEL
LIN {X 0,Y 350.158,Z 729.125,A -85,B 0,C 180,E1 14353.366,E2 14353.366} C_VEL
LIN {X 0,Y 350.838,Z 717.61,A -85,B 0,C 180,E1 14355.018,E2 14355.018} C_VEL
LIN {X 0,Y 351.319,Z 715.797,A -85,B 0,C 180,E1 14355.209,E2 14355.209} C_VEL
LIN {X 0,Y 360.563,Z 681.795,A -85,B 0,C 180,E1 14358.046,E2 14358.046} C_VEL
LIN {X 0,Y 363.516,Z 666.608,A -85,B 0,C 180,E1 14359.095,E2 14359.095} C_VEL
LIN {X 0,Y 353.113,Z 638.211,A -85,B 0,C 180,E1 14363.639,E2 14363.639} C_VEL
LIN {X 0,Y 340.693,Z 614.049,A -85,B 0,C 180,E1 14368.383,E2 14368.383} C_VEL
LIN {X 0,Y 328.698,Z 595.191,A -85,B 0,C 180,E1 14373.181,E2 14373.181} C_VEL
LIN {X 0,Y 320.555,Z 583.688,A -85,B 0,C 180,E1 14376.876,E2 14376.876} C_VEL
LIN {X 0,Y 316.1,Z 577.474,A -85,B 0,C 180,E1 14379.207,E2 14379.207} C_VEL
LIN {X 0,Y 312.367,Z 572.268,A -85,B 0,C 180,E1 14381.429,E2 14381.429} C_VEL
LIN {X 0,Y 310.671,Z 570.353,A -85,B 0,C 180,E1 14382.513,E2 14382.513} C_VEL
LIN {X 0,Y 306.742,Z 565.403,A -85,B 0,C 180,E1 14385.417,E2 14385.417} C_VEL
LIN {X 0,Y 306.543,Z 563.28,A -85,B 0,C 180,E1 14386.118,E2 14386.118} C_VEL
LIN {X 0,Y 307.12,Z 563.28,A -85,B 0,C 180,E1 14394.364,E2 14394.364} C_VEL
LIN {X 0,Y 307.57,Z 563.28,A -85,B 0,C 180,E1 14400.003,E2 14400.003} C_VEL
LIN {X 0,Y 306.929,Z 563.28,A -85,B 0,C 180,E1 14408.485,E2 14408.485} C_VEL
LIN {X 0,Y 306.592,Z 563.614,A -85,B 0,C 180,E1 14414.751,E2 14414.751} C_VEL
LIN {X 0,Y 308.388,Z 568.348,A -85,B 0,C 180,E1 14416.38,E2 14416.38} C_VEL
LIN {X 0,Y 312.43,Z 572.103,A -85,B 0,C 180,E1 14419.03,E2 14419.03} C_VEL
LIN {X 0,Y 316.113,Z 577.423,A -85,B 0,C 180,E1 14421.461,E2 14421.461} C_VEL
LIN {X 0,Y 318.728,Z 579.752,A -85,B 0,C 180,E1 14423.204,E2 14423.204} C_VEL
LIN {X 0,Y 322.234,Z 584.902,A -85,B 0,C 180,E1 14425.889,E2 14425.889} C_VEL
LIN {X 0,Y 325.486,Z 587.628,A -85,B 0,C 180,E1 14428.484,E2 14428.484} C_VEL
LIN {X 0,Y 329.694,Z 593.154,A -85,B 0,C 180,E1 14432.575,E2 14432.575} C_VEL
LIN {X 0,Y 332.444,Z 595.562,A -85,B 0,C 180,E1 14435.421,E2 14435.421} C_VEL
LIN {X 0,Y 336.199,Z 600.845,A -85,B 0,C 180,E1 14439.721,E2 14439.721} C_VEL
LIN {X 0,Y 339.205,Z 603.267,A -85,B 0,C 180,E1 14443.078,E2 14443.078} C_VEL
LIN {X 0,Y 343.387,Z 608.785,A -85,B 0,C 180,E1 14448.339,E2 14448.339} C_VEL
LIN {X 0,Y 346.691,Z 611.188,A -85,B 0,C 180,E1 14452.531,E2 14452.531} C_VEL
LIN {X 0,Y 350.045,Z 616.17,A -85,B 0,C 180,E1 14457.714,E2 14457.714} C_VEL
LIN {X 0,Y 354.252,Z 618.922,A -85,B 0,C 180,E1 14464.54,E2 14464.54} C_VEL
LIN {X 0,Y 356.864,Z 623.288,A -85,B 0,C 180,E1 14470.631,E2 14470.631} C_VEL
LIN {X 0,Y 359.019,Z 624.745,A -85,B 0,C 180,E1 14476.634,E2 14476.634} C_VEL
LIN {X 0,Y 360.545,Z 625.339,A -85,B 0,C 180,E1 14482.788,E2 14482.788} C_VEL
LIN {X 0,Y 361.163,Z 625.485,A -85,B 0,C 180,E1 14490.001,E2 14490.001} C_VEL
LIN {X 0,Y 360.539,Z 625.381,A -85,B 0,C 180,E1 14497.214,E2 14497.214} C_VEL
LIN {X 0,Y 358.875,Z 624.685,A -85,B 0,C 180,E1 14504,E2 14504} C_VEL
LIN {X 0,Y 356.297,Z 622.55,A -85,B 0,C 180,E1 14510.85,E2 14510.85} C_VEL
LIN {X 0,Y 353.763,Z 617.944,A -85,B 0,C 180,E1 14516.388,E2 14516.388} C_VEL
LIN {X 0,Y 349.621,Z 615.858,A -85,B 0,C 180,E1 14522.921,E2 14522.921} C_VEL
LIN {X 0,Y 346.45,Z 610.773,A -85,B 0,C 180,E1 14527.81,E2 14527.81} C_VEL
LIN {X 0,Y 341.112,Z 606.472,A -85,B 0,C 180,E1 14534.481,E2 14534.481} C_VEL
LIN {X 0,Y 338.332,Z 601.919,A -85,B 0,C 180,E1 14538.006,E2 14538.006} C_VEL
LIN {X 0,Y 333.64,Z 597.967,A -85,B 0,C 180,E1 14543.139,E2 14543.139} C_VEL
LIN {X 0,Y 331.256,Z 594.077,A -85,B 0,C 180,E1 14545.881,E2 14545.881} C_VEL
LIN {X 0,Y 326.372,Z 589.559,A -85,B 0,C 180,E1 14550.625,E2 14550.625} C_VEL
LIN {X 0,Y 324.305,Z 586.167,A -85,B 0,C 180,E1 14552.542,E2 14552.542} C_VEL
LIN {X 0,Y 319.606,Z 581.784,A -85,B 0,C 180,E1 14556.087,E2 14556.087} C_VEL
LIN {X 0,Y 317.461,Z 578.224,A -85,B 0,C 180,E1 14557.647,E2 14557.647} C_VEL
LIN {X 0,Y 312.984,Z 573.649,A -85,B 0,C 180,E1 14560.548,E2 14560.548} C_VEL
LIN {X 0,Y 311.4,Z 570.676,A -85,B 0,C 180,E1 14561.637,E2 14561.637} C_VEL
LIN {X 0,Y 306.845,Z 565.867,A -85,B 0,C 180,E1 14564.866,E2 14564.866} C_VEL
LIN {X 0,Y 306.446,Z 563.28,A -85,B 0,C 180,E1 14565.468,E2 14565.468} C_VEL
LIN {X 0,Y 306.945,Z 563.28,A -85,B 0,C 180,E1 14573.195,E2 14573.195} C_VEL
LIN {X 0,Y 307.539,Z 563.28,A -85,B 0,C 180,E1 14579.997,E2 14579.997} C_VEL
LIN {X 0,Y 306.942,Z 563.28,A -85,B 0,C 180,E1 14588.478,E2 14588.478} C_VEL
LIN {X 0,Y 306.658,Z 563.86,A -85,B 0,C 180,E1 14594.384,E2 14594.384} C_VEL
LIN {X 0,Y 308.582,Z 568.538,A -85,B 0,C 180,E1 14596.081,E2 14596.081} C_VEL
LIN {X 0,Y 312.271,Z 571.791,A -85,B 0,C 180,E1 14598.486,E2 14598.486} C_VEL
LIN {X 0,Y 315.942,Z 577.383,A -85,B 0,C 180,E1 14600.713,E2 14600.713} C_VEL
LIN {X 0,Y 318.197,Z 580.365,A -85,B 0,C 180,E1 14601.926,E2 14601.926} C_VEL
LIN {X 0,Y 327.51,Z 593.105,A -85,B 0,C 180,E1 14606.303,E2 14606.303} C_VEL
LIN {X 0,Y 341.358,Z 614.882,A -85,B 0,C 180,E1 14611.849,E2 14611.849} C_VEL
LIN {X 0,Y 353.796,Z 639.995,A -85,B 0,C 180,E1 14616.661,E2 14616.661} C_VEL
LIN {X 0,Y 363.502,Z 666.563,A -85,B 0,C 180,E1 14620.898,E2 14620.898} C_VEL
LIN {X 0,Y 354.756,Z 703.888,A -85,B 0,C 180,E1 14623.686,E2 14623.686} C_VEL
LIN {X 0,Y 344.436,Z 737.855,A -85,B 0,C 180,E1 14627.227,E2 14627.227} C_VEL
LIN {X 0,Y 332.979,Z 770.522,A -85,B 0,C 180,E1 14632.095,E2 14632.095} C_VEL
LIN {X 0,Y 323.194,Z 796.913,A -85,B 0,C 180,E1 14637.618,E2 14637.618} C_VEL
LIN {X 0,Y 315.418,Z 819.21,A -85,B 0,C 180,E1 14644.114,E2 14644.114} C_VEL
LIN {X 0,Y 310.467,Z 835.748,A -85,B 0,C 180,E1 14651.094,E2 14651.094} C_VEL
LIN {X 0,Y 308.32,Z 846.882,A -85,B 0,C 180,E1 14658.179,E2 14658.179} C_VEL
LIN {X 0,Y 307.696,Z 852.257,A -85,B 0,C 180,E1 14664.37,E2 14664.37} C_VEL
LIN {X 0,Y 307.773,Z 853.874,A -85,B 0,C 180,E1 14669.999,E2 14669.999} C_VEL
LIN {X 0,Y 307.73,Z 851.301,A -85,B 0,C 180,E1 14677.04,E2 14677.04} C_VEL
LIN {X 0,Y 308.817,Z 843.796,A -85,B 0,C 180,E1 14684.14,E2 14684.14} C_VEL
LIN {X 0,Y 311.833,Z 830.806,A -85,B 0,C 180,E1 14691.279,E2 14691.279} C_VEL
LIN {X 0,Y 317.964,Z 811.727,A -85,B 0,C 180,E1 14698.331,E2 14698.331} C_VEL
LIN {X 0,Y 327.102,Z 786.363,A -85,B 0,C 180,E1 14704.811,E2 14704.811} C_VEL
LIN {X 0,Y 337.012,Z 759.283,A -85,B 0,C 180,E1 14709.78,E2 14709.78} C_VEL
LIN {X 0,Y 348.557,Z 725.083,A -85,B 0,C 180,E1 14714.255,E2 14714.255} C_VEL
LIN {X 0,Y 351.319,Z 715.797,A -85,B 0,C 180,E1 14715.209,E2 14715.209} C_VEL
LIN {X 0,Y 352.562,Z 701.945,A -85,B 0,C 180,E1 14716.946,E2 14716.946} C_VEL
LIN {X 0,Y 353.682,Z 687.604,A -85,B 0,C 180,E1 14718.56,E2 14718.56} C_VEL
LIN {X 0,Y 357.674,Z 669.965,A -85,B 0,C 180,E1 14719.814,E2 14719.814} C_VEL
LIN {X 0,Y 347.925,Z 642.44,A -85,B 0,C 180,E1 14724.412,E2 14724.412} C_VEL
LIN {X 0,Y 336.456,Z 619.096,A -85,B 0,C 180,E1 14729.215,E2 14729.215} C_VEL
LIN {X 0,Y 323.654,Z 598.163,A -85,B 0,C 180,E1 14734.793,E2 14734.793} C_VEL
LIN {X 0,Y 313.939,Z 584.657,A -85,B 0,C 180,E1 14739.792,E2 14739.792} C_VEL
LIN {X 0,Y 309.21,Z 577.967,A -85,B 0,C 180,E1 14742.794,E2 14742.794} C_VEL
LIN {X 0,Y 305.074,Z 572.649,A -85,B 0,C 180,E1 14745.958,E2 14745.958} C_VEL
LIN {X 0,Y 304.272,Z 570.846,A -85,B 0,C 180,E1 14746.743,E2 14746.743} C_VEL
LIN {X 0,Y 299.467,Z 566.023,A -85,B 0,C 180,E1 14752.129,E2 14752.129} C_VEL
LIN {X 0,Y 299.078,Z 563.28,A -85,B 0,C 180,E1 14753.485,E2 14753.485} C_VEL
LIN {X 0,Y 299.675,Z 563.28,A -85,B 0,C 180,E1 14760.003,E2 14760.003} C_VEL
LIN {X 0,Y 299.053,Z 563.921,A -85,B 0,C 180,E1 14767.341,E2 14767.341} C_VEL
LIN {X 0,Y 301.705,Z 569.311,A -85,B 0,C 180,E1 14771.296,E2 14771.296} C_VEL
LIN {X 0,Y 304.963,Z 571.917,A -85,B 0,C 180,E1 14774.327,E2 14774.327} C_VEL
LIN {X 0,Y 308.601,Z 577.552,A -85,B 0,C 180,E1 14777.247,E2 14777.247} C_VEL
LIN {X 0,Y 310.768,Z 579.917,A -85,B 0,C 180,E1 14778.676,E2 14778.676} C_VEL
LIN {X 0,Y 315.051,Z 585.335,A -85,B 0,C 180,E1 14781.468,E2 14781.468} C_VEL
LIN {X 0,Y 317.351,Z 588.008,A -85,B 0,C 180,E1 14783.051,E2 14783.051} C_VEL
LIN {X 0,Y 321.546,Z 593.091,A -85,B 0,C 180,E1 14786.257,E2 14786.257} C_VEL
LIN {X 0,Y 324.131,Z 595.639,A -85,B 0,C 180,E1 14788.375,E2 14788.375} C_VEL
LIN {X 0,Y 328.642,Z 601.045,A -85,B 0,C 180,E1 14792.629,E2 14792.629} C_VEL
LIN {X 0,Y 331.223,Z 603.394,A -85,B 0,C 180,E1 14795.23,E2 14795.23} C_VEL
LIN {X 0,Y 335.338,Z 608.765,A -85,B 0,C 180,E1 14799.844,E2 14799.844} C_VEL
LIN {X 0,Y 338.096,Z 611.17,A -85,B 0,C 180,E1 14802.956,E2 14802.956} C_VEL
LIN {X 0,Y 342.412,Z 616.639,A -85,B 0,C 180,E1 14808.341,E2 14808.341} C_VEL
LIN {X 0,Y 345.546,Z 618.927,A -85,B 0,C 180,E1 14812.312,E2 14812.312} C_VEL
LIN {X 0,Y 348.999,Z 623.947,A -85,B 0,C 180,E1 14817.605,E2 14817.605} C_VEL
LIN {X 0,Y 353.217,Z 626.835,A -85,B 0,C 180,E1 14824.46,E2 14824.46} C_VEL
LIN {X 0,Y 355.973,Z 631.182,A -85,B 0,C 180,E1 14830.787,E2 14830.787} C_VEL
LIN {X 0,Y 358.088,Z 632.58,A -85,B 0,C 180,E1 14836.749,E2 14836.749} C_VEL
LIN {X 0,Y 359.576,Z 633.178,A -85,B 0,C 180,E1 14842.768,E2 14842.768} C_VEL
LIN {X 0,Y 360.201,Z 633.325,A -85,B 0,C 180,E1 14850.001,E2 14850.001} C_VEL
LIN {X 0,Y 359.571,Z 633.22,A -85,B 0,C 180,E1 14857.234,E2 14857.234} C_VEL
LIN {X 0,Y 357.889,Z 632.486,A -85,B 0,C 180,E1 14864.116,E2 14864.116} C_VEL
LIN {X 0,Y 355.246,Z 630.308,A -85,B 0,C 180,E1 14871.054,E2 14871.054} C_VEL
LIN {X 0,Y 352.387,Z 625.679,A -85,B 0,C 180,E1 14877.13,E2 14877.13} C_VEL
LIN {X 0,Y 348.073,Z 623.141,A -85,B 0,C 180,E1 14883.817,E2 14883.817} C_VEL
LIN {X 0,Y 344.29,Z 617.51,A -85,B 0,C 180,E1 14889.405,E2 14889.405} C_VEL
LIN {X 0,Y 339.599,Z 613.688,A -85,B 0,C 180,E1 14895.147,E2 14895.147} C_VEL
LIN {X 0,Y 337.018,Z 609.606,A -85,B 0,C 180,E1 14898.37,E2 14898.37} C_VEL
LIN {X 0,Y 332.317,Z 605.474,A -85,B 0,C 180,E1 14903.501,E2 14903.501} C_VEL
LIN {X 0,Y 329.869,Z 601.785,A -85,B 0,C 180,E1 14906.211,E2 14906.211} C_VEL
LIN {X 0,Y 324.709,Z 596.889,A -85,B 0,C 180,E1 14911.052,E2 14911.052} C_VEL
LIN {X 0,Y 322.292,Z 593.563,A -85,B 0,C 180,E1 14913.182,E2 14913.182} C_VEL
LIN {X 0,Y 317.732,Z 588.819,A -85,B 0,C 180,E1 14916.643,E2 14916.643} C_VEL
LIN {X 0,Y 315.622,Z 585.655,A -85,B 0,C 180,E1 14918.186,E2 14918.186} C_VEL
LIN {X 0,Y 310.995,Z 580.544,A -85,B 0,C 180,E1 14921.154,E2 14921.154} C_VEL
LIN {X 0,Y 309.378,Z 578.094,A -85,B 0,C 180,E1 14922.248,E2 14922.248} C_VEL
LIN {X 0,Y 305.006,Z 572.526,A -85,B 0,C 180,E1 14925.584,E2 14925.584} C_VEL
LIN {X 0,Y 304.193,Z 570.846,A -85,B 0,C 180,E1 14926.368,E2 14926.368} C_VEL
LIN {X 0,Y 299.491,Z 565.979,A -85,B 0,C 180,E1 14931.668,E2 14931.668} C_VEL
LIN {X 0,Y 299.054,Z 563.28,A -85,B 0,C 180,E1 14933.237,E2 14933.237} C_VEL
LIN {X 0,Y 299.649,Z 563.28,A -85,B 0,C 180,E1 14939.997,E2 14939.997} C_VEL
LIN {X 0,Y 299.087,Z 563.994,A -85,B 0,C 180,E1 14946.97,E2 14946.97} C_VEL
LIN {X 0,Y 301.874,Z 569.426,A -85,B 0,C 180,E1 14951.036,E2 14951.036} C_VEL
LIN {X 0,Y 304.958,Z 571.683,A -85,B 0,C 180,E1 14953.864,E2 14953.864} C_VEL
LIN {X 0,Y 308.189,Z 577.217,A -85,B 0,C 180,E1 14956.532,E2 14956.532} C_VEL
LIN {X 0,Y 310.597,Z 579.727,A -85,B 0,C 180,E1 14958.131,E2 14958.131} C_VEL
LIN {X 0,Y 316.719,Z 588.549,A -85,B 0,C 180,E1 14961.758,E2 14961.758} C_VEL
LIN {X 0,Y 325.066,Z 600.27,A -85,B 0,C 180,E1 14965.862,E2 14965.862} C_VEL
LIN {X 0,Y 338.081,Z 621.647,A -85,B 0,C 180,E1 14971.424,E2 14971.424} C_VEL
LIN {X 0,Y 349.751,Z 646.871,A -85,B 0,C 180,E1 14976.384,E2 14976.384} C_VEL
LIN {X 0,Y 357.673,Z 671.246,A -85,B 0,C 180,E1 14980.324,E2 14980.324} C_VEL
LIN {X 0,Y 347.422,Z 710.038,A -85,B 0,C 180,E1 14983.297,E2 14983.297} C_VEL
LIN {X 0,Y 336.078,Z 744.583,A -85,B 0,C 180,E1 14987.223,E2 14987.223} C_VEL
LIN {X 0,Y 325.213,Z 773.88,A -85,B 0,C 180,E1 14991.875,E2 14991.875} C_VEL
LIN {X 0,Y 314.38,Z 801.758,A -85,B 0,C 180,E1 14998.128,E2 14998.128} C_VEL
LIN {X 0,Y 306.631,Z 823.062,A -85,B 0,C 180,E1 15005.016,E2 15005.016} C_VEL
LIN {X 0,Y 302.423,Z 837.104,A -85,B 0,C 180,E1 15011.438,E2 15011.438} C_VEL
LIN {X 0,Y 300.384,Z 847.191,A -85,B 0,C 180,E1 15018.406,E2 15018.406} C_VEL
LIN {X 0,Y 299.796,Z 852.011,A -85,B 0,C 180,E1 15024.221,E2 15024.221} C_VEL
LIN {X 0,Y 299.889,Z 853.629,A -85,B 0,C 180,E1 15029.999,E2 15029.999} C_VEL
LIN {X 0,Y 299.869,Z 851.055,A -85,B 0,C 180,E1 15037.226,E2 15037.226} C_VEL
LIN {X 0,Y 301.003,Z 843.546,A -85,B 0,C 180,E1 15044.515,E2 15044.515} C_VEL
LIN {X 0,Y 304.271,Z 830.554,A -85,B 0,C 180,E1 15051.835,E2 15051.835} C_VEL
LIN {X 0,Y 310.832,Z 811.319,A -85,B 0,C 180,E1 15059.098,E2 15059.098} C_VEL
LIN {X 0,Y 320.428,Z 786.109,A -85,B 0,C 180,E1 15065.645,E2 15065.645} C_VEL
LIN {X 0,Y 331.053,Z 758.221,A -85,B 0,C 180,E1 15070.811,E2 15070.811} C_VEL
LIN {X 0,Y 343.026,Z 724.212,A -85,B 0,C 180,E1 15075.267,E2 15075.267} C_VEL
LIN {X 0,Y 353.682,Z 687.604,A -85,B 0,C 180,E1 15078.56,E2 15078.56} C_VEL
LIN {X 0,Y 354.322,Z 680.27,A -85,B 0,C 180,E1 15079.318,E2 15079.318} C_VEL
LIN {X 0,Y 353.028,Z 673.837,A -85,B 0,C 180,E1 15080.285,E2 15080.285} C_VEL
LIN {X 0,Y 348.438,Z 661.857,A -85,B 0,C 180,E1 15082.45,E2 15082.45} C_VEL
LIN {X 0,Y 337.933,Z 635.327,A -85,B 0,C 180,E1 15087.483,E2 15087.483} C_VEL
LIN {X 0,Y 325.127,Z 611.564,A -85,B 0,C 180,E1 15093.288,E2 15093.288} C_VEL
LIN {X 0,Y 312.788,Z 592.585,A -85,B 0,C 180,E1 15099.807,E2 15099.807} C_VEL
LIN {X 0,Y 307.239,Z 585.288,A -85,B 0,C 180,E1 15103.416,E2 15103.416} C_VEL
LIN {X 0,Y 303.344,Z 579.539,A -85,B 0,C 180,E1 15106.61,E2 15106.61} C_VEL
LIN {X 0,Y 298.02,Z 572.753,A -85,B 0,C 180,E1 15113.005,E2 15113.005} C_VEL
LIN {X 0,Y 297.528,Z 570.986,A -85,B 0,C 180,E1 15114.181,E2 15114.181} C_VEL
LIN {X 0,Y 297.786,Z 571.104,A -85,B 0,C 180,E1 15126.733,E2 15126.733} C_VEL
LIN {X 0,Y 300.326,Z 576.858,A -85,B 0,C 180,E1 15130.864,E2 15130.864} C_VEL
LIN {X 0,Y 303.476,Z 579.64,A -85,B 0,C 180,E1 15133.94,E2 15133.94} C_VEL
LIN {X 0,Y 307.873,Z 585.685,A -85,B 0,C 180,E1 15137.473,E2 15137.473} C_VEL
LIN {X 0,Y 313.362,Z 592.919,A -85,B 0,C 180,E1 15141.189,E2 15141.189} C_VEL
LIN {X 0,Y 315.882,Z 596.201,A -85,B 0,C 180,E1 15142.991,E2 15142.991} C_VEL
LIN {X 0,Y 320.673,Z 601.157,A -85,B 0,C 180,E1 15146.61,E2 15146.61} C_VEL
LIN {X 0,Y 326.726,Z 608.418,A -85,B 0,C 180,E1 15152.032,E2 15152.032} C_VEL
LIN {X 0,Y 329.892,Z 611.178,A -85,B 0,C 180,E1 15155.054,E2 15155.054} C_VEL
LIN {X 0,Y 334.1,Z 616.475,A -85,B 0,C 180,E1 15159.622,E2 15159.622} C_VEL
LIN {X 0,Y 336.92,Z 618.946,A -85,B 0,C 180,E1 15162.74,E2 15162.74} C_VEL
LIN {X 0,Y 341.166,Z 624.334,A -85,B 0,C 180,E1 15168.03,E2 15168.03} C_VEL
LIN {X 0,Y 344.443,Z 626.76,A -85,B 0,C 180,E1 15172.17,E2 15172.17} C_VEL
LIN {X 0,Y 348.172,Z 631.935,A -85,B 0,C 180,E1 15177.82,E2 15177.82} C_VEL
LIN {X 0,Y 352.14,Z 634.599,A -85,B 0,C 180,E1 15184.293,E2 15184.293} C_VEL
LIN {X 0,Y 354.876,Z 638.945,A -85,B 0,C 180,E1 15190.518,E2 15190.518} C_VEL
LIN {X 0,Y 357.197,Z 640.461,A -85,B 0,C 180,E1 15197.009,E2 15197.009} C_VEL
LIN {X 0,Y 358.61,Z 641,A -85,B 0,C 180,E1 15202.749,E2 15202.749} C_VEL
LIN {X 0,Y 359.238,Z 641.165,A -85,B 0,C 180,E1 15210.001,E2 15210.001} C_VEL
LIN {X 0,Y 358.602,Z 641.059,A -85,B 0,C 180,E1 15217.254,E2 15217.254} C_VEL
LIN {X 0,Y 357.041,Z 640.421,A -85,B 0,C 180,E1 15223.564,E2 15223.564} C_VEL
LIN {X 0,Y 354.543,Z 638.503,A -85,B 0,C 180,E1 15230.325,E2 15230.325} C_VEL
LIN {X 0,Y 351.949,Z 633.991,A -85,B 0,C 180,E1 15236.113,E2 15236.113} C_VEL
LIN {X 0,Y 347.632,Z 631.572,A -85,B 0,C 180,E1 15242.984,E2 15242.984} C_VEL
LIN {X 0,Y 344.183,Z 626.359,A -85,B 0,C 180,E1 15248.182,E2 15248.182} C_VEL
LIN {X 0,Y 338.828,Z 621.889,A -85,B 0,C 180,E1 15254.899,E2 15254.899} C_VEL
LIN {X 0,Y 335.911,Z 617.405,A -85,B 0,C 180,E1 15258.496,E2 15258.496} C_VEL
LIN {X 0,Y 331.035,Z 613.24,A -85,B 0,C 180,E1 15263.656,E2 15263.656} C_VEL
LIN {X 0,Y 328.321,Z 609.402,A -85,B 0,C 180,E1 15266.525,E2 15266.525} C_VEL
LIN {X 0,Y 322.864,Z 604.248,A -85,B 0,C 180,E1 15271.468,E2 15271.468} C_VEL
LIN {X 0,Y 320.434,Z 601.048,A -85,B 0,C 180,E1 15273.568,E2 15273.568} C_VEL
LIN {X 0,Y 315.675,Z 595.878,A -85,B 0,C 180,E1 15277.17,E2 15277.17} C_VEL
LIN {X 0,Y 313.348,Z 592.875,A -85,B 0,C 180,E1 15278.83,E2 15278.83} C_VEL
LIN {X 0,Y 308.709,Z 586.874,A -85,B 0,C 180,E1 15281.933,E2 15281.933} C_VEL
LIN {X 0,Y 303.362,Z 579.66,A -85,B 0,C 180,E1 15286.147,E2 15286.147} C_VEL
LIN {X 0,Y 297.996,Z 572.606,A -85,B 0,C 180,E1 15292.633,E2 15292.633} C_VEL
LIN {X 0,Y 297.307,Z 570.951,A -85,B 0,C 180,E1 15294.171,E2 15294.171} C_VEL
LIN {X 0,Y 297.823,Z 571.115,A -85,B 0,C 180,E1 15306.36,E2 15306.36} C_VEL
LIN {X 0,Y 300.386,Z 576.871,A -85,B 0,C 180,E1 15310.489,E2 15310.489} C_VEL
LIN {X 0,Y 303.541,Z 579.754,A -85,B 0,C 180,E1 15313.564,E2 15313.564} C_VEL
LIN {X 0,Y 307.757,Z 585.565,A -85,B 0,C 180,E1 15316.922,E2 15316.922} C_VEL
LIN {X 0,Y 315.522,Z 597.14,A -85,B 0,C 180,E1 15321.844,E2 15321.844} C_VEL
LIN {X 0,Y 325.689,Z 612.573,A -85,B 0,C 180,E1 15326.985,E2 15326.985} C_VEL
LIN {X 0,Y 338.056,Z 635.502,A -85,B 0,C 180,E1 15332.564,E2 15332.564} C_VEL
LIN {X 0,Y 348.871,Z 663.324,A -85,B 0,C 180,E1 15337.788,E2 15337.788} C_VEL
LIN {X 0,Y 351.68,Z 674.555,A -85,B 0,C 180,E1 15339.563,E2 15339.563} C_VEL
LIN {X 0,Y 341.429,Z 711.443,A -85,B 0,C 180,E1 15342.476,E2 15342.476} C_VEL
LIN {X 0,Y 329.328,Z 746.657,A -85,B 0,C 180,E1 15346.581,E2 15346.581} C_VEL
LIN {X 0,Y 318.04,Z 775.54,A -85,B 0,C 180,E1 15351.349,E2 15351.349} C_VEL
LIN {X 0,Y 307.458,Z 801.503,A -85,B 0,C 180,E1 15357.323,E2 15357.323} C_VEL
LIN {X 0,Y 299.747,Z 821.388,A -85,B 0,C 180,E1 15363.797,E2 15363.797} C_VEL
LIN {X 0,Y 294.721,Z 836.852,A -85,B 0,C 180,E1 15370.935,E2 15370.935} C_VEL
LIN {X 0,Y 292.456,Z 847.447,A -85,B 0,C 180,E1 15378.605,E2 15378.605} C_VEL
LIN {X 0,Y 291.899,Z 851.764,A -85,B 0,C 180,E1 15384.064,E2 15384.064} C_VEL
LIN {X 0,Y 291.989,Z 853.384,A -85,B 0,C 180,E1 15389.999,E2 15389.999} C_VEL
LIN {X 0,Y 291.976,Z 850.808,A -85,B 0,C 180,E1 15397.422,E2 15397.422} C_VEL
LIN {X 0,Y 293.218,Z 843.296,A -85,B 0,C 180,E1 15404.91,E2 15404.91} C_VEL
LIN {X 0,Y 296.743,Z 830.301,A -85,B 0,C 180,E1 15412.418,E2 15412.418} C_VEL
LIN {X 0,Y 303.639,Z 811.218,A -85,B 0,C 180,E1 15419.799,E2 15419.799} C_VEL
LIN {X 0,Y 313.799,Z 785.854,A -85,B 0,C 180,E1 15426.518,E2 15426.518} C_VEL
LIN {X 0,Y 325.02,Z 757.706,A -85,B 0,C 180,E1 15431.791,E2 15431.791} C_VEL
LIN {X 0,Y 337.391,Z 723.961,A -85,B 0,C 180,E1 15436.242,E2 15436.242} C_VEL
LIN {X 0,Y 348.077,Z 688.678,A -85,B 0,C 180,E1 15439.446,E2 15439.446} C_VEL
LIN {X 0,Y 351.613,Z 672.56,A -85,B 0,C 180,E1 15440.673,E2 15440.673} C_VEL
LIN {X 0,Y 348.438,Z 661.857,A -85,B 0,C 180,E1 15442.45,E2 15442.45} C_VEL
LIN {X 0,Y 343.984,Z 654.918,A -85,B 0,C 180,E1 15444.139,E2 15444.139} C_VEL
LIN {X 0,Y 335.434,Z 645.167,A -85,B 0,C 180,E1 15447.17,E2 15447.17} C_VEL
LIN {X 0,Y 324.496,Z 622.87,A -85,B 0,C 180,E1 15452.549,E2 15452.549} C_VEL
LIN {X 0,Y 313.956,Z 605.186,A -85,B 0,C 180,E1 15458.226,E2 15458.226} C_VEL
LIN {X 0,Y 308.845,Z 597.972,A -85,B 0,C 180,E1 15461.382,E2 15461.382} C_VEL
LIN {X 0,Y 305.463,Z 592.704,A -85,B 0,C 180,E1 15463.87,E2 15463.87} C_VEL
LIN {X 0,Y 300.793,Z 585.907,A -85,B 0,C 180,E1 15468.06,E2 15468.06} C_VEL
LIN {X 0,Y 296.82,Z 580.235,A -85,B 0,C 180,E1 15473.435,E2 15473.435} C_VEL
LIN {X 0,Y 296.57,Z 578.831,A -85,B 0,C 180,E1 15474.162,E2 15474.162} C_VEL
LIN {X 0,Y 296.632,Z 578.853,A -85,B 0,C 180,E1 15486.392,E2 15486.392} C_VEL
LIN {X 0,Y 299.341,Z 584.778,A -85,B 0,C 180,E1 15490.9,E2 15490.9} C_VEL
LIN {X 0,Y 302.028,Z 587.505,A -85,B 0,C 180,E1 15493.639,E2 15493.639} C_VEL
LIN {X 0,Y 307.514,Z 595.83,A -85,B 0,C 180,E1 15498.233,E2 15498.233} C_VEL
LIN {X 0,Y 313.769,Z 603.452,A -85,B 0,C 180,E1 15502.569,E2 15502.569} C_VEL
LIN {X 0,Y 318.807,Z 608.759,A -85,B 0,C 180,E1 15506.362,E2 15506.362} C_VEL
LIN {X 0,Y 325.234,Z 616.21,A -85,B 0,C 180,E1 15512.032,E2 15512.032} C_VEL
LIN {X 0,Y 328.34,Z 618.965,A -85,B 0,C 180,E1 15514.898,E2 15514.898} C_VEL
LIN {X 0,Y 333.023,Z 624.364,A -85,B 0,C 180,E1 15519.775,E2 15519.775} C_VEL
LIN {X 0,Y 335.653,Z 626.823,A -85,B 0,C 180,E1 15522.621,E2 15522.621} C_VEL
LIN {X 0,Y 340.165,Z 632.185,A -85,B 0,C 180,E1 15528.029,E2 15528.029} C_VEL
LIN {X 0,Y 343.309,Z 634.523,A -85,B 0,C 180,E1 15531.978,E2 15531.978} C_VEL
LIN {X 0,Y 347.011,Z 639.644,A -85,B 0,C 180,E1 15537.548,E2 15537.548} C_VEL
LIN {X 0,Y 351.047,Z 642.333,A -85,B 0,C 180,E1 15544.089,E2 15544.089} C_VEL
LIN {X 0,Y 353.797,Z 646.653,A -85,B 0,C 180,E1 15550.253,E2 15550.253} C_VEL
LIN {X 0,Y 356.072,Z 648.219,A -85,B 0,C 180,E1 15556.396,E2 15556.396} C_VEL
LIN {X 0,Y 357.643,Z 648.827,A -85,B 0,C 180,E1 15562.729,E2 15562.729} C_VEL
LIN {X 0,Y 358.275,Z 649.005,A -85,B 0,C 180,E1 15570.001,E2 15570.001} C_VEL
LIN {X 0,Y 357.635,Z 648.884,A -85,B 0,C 180,E1 15577.273,E2 15577.273} C_VEL
LIN {X 0,Y 356.068,Z 648.257,A -85,B 0,C 180,E1 15583.602,E2 15583.602} C_VEL
LIN {X 0,Y 353.64,Z 646.439,A -85,B 0,C 180,E1 15590.151,E2 15590.151} C_VEL
LIN {X 0,Y 350.94,Z 641.971,A -85,B 0,C 180,E1 15596.147,E2 15596.147} C_VEL
LIN {X 0,Y 346.59,Z 639.373,A -85,B 0,C 180,E1 15603.097,E2 15603.097} C_VEL
LIN {X 0,Y 342.992,Z 633.965,A -85,B 0,C 180,E1 15608.478,E2 15608.478} C_VEL
LIN {X 0,Y 337.61,Z 629.662,A -85,B 0,C 180,E1 15615.024,E2 15615.024} C_VEL
LIN {X 0,Y 334.233,Z 624.995,A -85,B 0,C 180,E1 15619.018,E2 15619.018} C_VEL
LIN {X 0,Y 329.132,Z 620.412,A -85,B 0,C 180,E1 15624.214,E2 15624.214} C_VEL
LIN {X 0,Y 326.568,Z 617.006,A -85,B 0,C 180,E1 15626.831,E2 15626.831} C_VEL
LIN {X 0,Y 320.872,Z 611.581,A -85,B 0,C 180,E1 15631.849,E2 15631.849} C_VEL
LIN {X 0,Y 318.047,Z 608.377,A -85,B 0,C 180,E1 15634.178,E2 15634.178} C_VEL
LIN {X 0,Y 313.261,Z 602.532,A -85,B 0,C 180,E1 15637.83,E2 15637.83} C_VEL
LIN {X 0,Y 306.865,Z 594.518,A -85,B 0,C 180,E1 15642.283,E2 15642.283} C_VEL
LIN {X 0,Y 301.662,Z 586.792,A -85,B 0,C 180,E1 15646.712,E2 15646.712} C_VEL
LIN {X 0,Y 296.869,Z 580.438,A -85,B 0,C 180,E1 15652.88,E2 15652.88} C_VEL
LIN {X 0,Y 296.349,Z 578.793,A -85,B 0,C 180,E1 15654.152,E2 15654.152} C_VEL
LIN {X 0,Y 296.655,Z 578.963,A -85,B 0,C 180,E1 15666.019,E2 15666.019} C_VEL
LIN {X 0,Y 299.588,Z 584.949,A -85,B 0,C 180,E1 15670.701,E2 15670.701} C_VEL
LIN {X 0,Y 302.127,Z 587.621,A -85,B 0,C 180,E1 15673.261,E2 15673.261} C_VEL
LIN {X 0,Y 307.376,Z 595.558,A -85,B 0,C 180,E1 15677.599,E2 15677.599} C_VEL
LIN {X 0,Y 315.394,Z 607.163,A -85,B 0,C 180,E1 15682.598,E2 15682.598} C_VEL
LIN {X 0,Y 326.663,Z 626.831,A -85,B 0,C 180,E1 15688.538,E2 15688.538} C_VEL
LIN {X 0,Y 337.079,Z 649.139,A -85,B 0,C 180,E1 15693.638,E2 15693.638} C_VEL
LIN {X 0,Y 345.861,Z 676.052,A -85,B 0,C 180,E1 15698.588,E2 15698.588} C_VEL
LIN {X 0,Y 335.541,Z 712.648,A -85,B 0,C 180,E1 15701.61,E2 15701.61} C_VEL
LIN {X 0,Y 323.035,Z 747.659,A -85,B 0,C 180,E1 15705.767,E2 15705.767} C_VEL
LIN {X 0,Y 310.764,Z 777.49,A -85,B 0,C 180,E1 15710.856,E2 15710.856} C_VEL
LIN {X 0,Y 300.061,Z 802.536,A -85,B 0,C 180,E1 15716.843,E2 15716.843} C_VEL
LIN {X 0,Y 291.202,Z 824.464,A -85,B 0,C 180,E1 15724.43,E2 15724.43} C_VEL
LIN {X 0,Y 286.519,Z 838.529,A -85,B 0,C 180,E1 15731.577,E2 15731.577} C_VEL
LIN {X 0,Y 284.416,Z 848.578,A -85,B 0,C 180,E1 15739.729,E2 15739.729} C_VEL
LIN {X 0,Y 283.965,Z 852.728,A -85,B 0,C 180,E1 15746.952,E2 15746.952} C_VEL
LIN {X 0,Y 283.979,Z 852.729,A -85,B 0,C 180,E1 15753.045,E2 15753.045} C_VEL
LIN {X 0,Y 284.377,Z 848.603,A -85,B 0,C 180,E1 15760.245,E2 15760.245} C_VEL
LIN {X 0,Y 286.613,Z 838.536,A -85,B 0,C 180,E1 15768.414,E2 15768.414} C_VEL
LIN {X 0,Y 291.752,Z 823.182,A -85,B 0,C 180,E1 15776.079,E2 15776.079} C_VEL
LIN {X 0,Y 300.116,Z 802.548,A -85,B 0,C 180,E1 15783.146,E2 15783.146} C_VEL
LIN {X 0,Y 311.423,Z 775.812,A -85,B 0,C 180,E1 15789.491,E2 15789.491} C_VEL
LIN {X 0,Y 323.447,Z 746.422,A -85,B 0,C 180,E1 15794.41,E2 15794.41} C_VEL
LIN {X 0,Y 336.016,Z 711.214,A -85,B 0,C 180,E1 15798.538,E2 15798.538} C_VEL
LIN {X 0,Y 345.882,Z 676.056,A -85,B 0,C 180,E1 15801.407,E2 15801.407} C_VEL
LIN {X 0,Y 337.722,Z 650.724,A -85,B 0,C 180,E1 15806.05,E2 15806.05} C_VEL
LIN {X 0,Y 335.434,Z 645.167,A -85,B 0,C 180,E1 15807.17,E2 15807.17} C_VEL
LIN {X 0,Y 330.758,Z 639.411,A -85,B 0,C 180,E1 15809.033,E2 15809.033} C_VEL
LIN {X 0,Y 322.332,Z 631.884,A -85,B 0,C 180,E1 15812.378,E2 15812.378} C_VEL
LIN {X 0,Y 311.8,Z 612.776,A -85,B 0,C 180,E1 15818.441,E2 15818.441} C_VEL
LIN {X 0,Y 303.576,Z 600.067,A -85,B 0,C 180,E1 15824.322,E2 15824.322} C_VEL
LIN {X 0,Y 299.338,Z 593.56,A -85,B 0,C 180,E1 15828.37,E2 15828.37} C_VEL
LIN {X 0,Y 295.622,Z 587.746,A -85,B 0,C 180,E1 15833.831,E2 15833.831} C_VEL
LIN {X 0,Y 294.537,Z 586.27,A -85,B 0,C 180,E1 15836.699,E2 15836.699} C_VEL
LIN {X 0,Y 295.52,Z 587.146,A -85,B 0,C 180,E1 15846.324,E2 15846.324} C_VEL
LIN {X 0,Y 298.837,Z 593.261,A -85,B 0,C 180,E1 15851.656,E2 15851.656} C_VEL
LIN {X 0,Y 300.494,Z 595.473,A -85,B 0,C 180,E1 15853.433,E2 15853.433} C_VEL
LIN {X 0,Y 305.67,Z 603.663,A -85,B 0,C 180,E1 15858.067,E2 15858.067} C_VEL
LIN {X 0,Y 311.636,Z 610.995,A -85,B 0,C 180,E1 15862.298,E2 15862.298} C_VEL
LIN {X 0,Y 317.01,Z 616.449,A -85,B 0,C 180,E1 15866.317,E2 15866.317} C_VEL
LIN {X 0,Y 323.374,Z 623.808,A -85,B 0,C 180,E1 15871.844,E2 15871.844} C_VEL
LIN {X 0,Y 326.605,Z 626.719,A -85,B 0,C 180,E1 15874.775,E2 15874.775} C_VEL
LIN {X 0,Y 331.551,Z 632.132,A -85,B 0,C 180,E1 15879.764,E2 15879.764} C_VEL
LIN {X 0,Y 334.208,Z 634.776,A -85,B 0,C 180,E1 15882.634,E2 15882.634} C_VEL
LIN {X 0,Y 338.958,Z 640.004,A -85,B 0,C 180,E1 15888.105,E2 15888.105} C_VEL
LIN {X 0,Y 342.052,Z 642.367,A -85,B 0,C 180,E1 15891.858,E2 15891.858} C_VEL
LIN {X 0,Y 345.964,Z 647.496,A -85,B 0,C 180,E1 15897.59,E2 15897.59} C_VEL
LIN {X 0,Y 350.022,Z 650.26,A -85,B 0,C 180,E1 15904.038,E2 15904.038} C_VEL
LIN {X 0,Y 352.805,Z 654.494,A -85,B 0,C 180,E1 15910.221,E2 15910.221} C_VEL
LIN {X 0,Y 355.042,Z 656.028,A -85,B 0,C 180,E1 15916.088,E2 15916.088} C_VEL
LIN {X 0,Y 356.677,Z 656.641,A -85,B 0,C 180,E1 15922.709,E2 15922.709} C_VEL
LIN {X 0,Y 357.313,Z 656.84,A -85,B 0,C 180,E1 15930.001,E2 15930.001} C_VEL
LIN {X 0,Y 356.666,Z 656.723,A -85,B 0,C 180,E1 15937.293,E2 15937.293} C_VEL
LIN {X 0,Y 355.038,Z 656.052,A -85,B 0,C 180,E1 15943.913,E2 15943.913} C_VEL
LIN {X 0,Y 352.471,Z 654.034,A -85,B 0,C 180,E1 15950.685,E2 15950.685} C_VEL
LIN {X 0,Y 349.357,Z 649.146,A -85,B 0,C 180,E1 15957.302,E2 15957.302} C_VEL
LIN {X 0,Y 345.013,Z 646.716,A -85,B 0,C 180,E1 15963.793,E2 15963.793} C_VEL
LIN {X 0,Y 340.532,Z 640.752,A -85,B 0,C 180,E1 15970.101,E2 15970.101} C_VEL
LIN {X 0,Y 335.447,Z 636.534,A -85,B 0,C 180,E1 15975.964,E2 15975.964} C_VEL
LIN {X 0,Y 332.392,Z 632.523,A -85,B 0,C 180,E1 15979.433,E2 15979.433} C_VEL
LIN {X 0,Y 327.192,Z 627.77,A -85,B 0,C 180,E1 15984.59,E2 15984.59} C_VEL
LIN {X 0,Y 324.474,Z 624.485,A -85,B 0,C 180,E1 15987.232,E2 15987.232} C_VEL
LIN {X 0,Y 318.59,Z 618.714,A -85,B 0,C 180,E1 15992.302,E2 15992.302} C_VEL
LIN {X 0,Y 314.665,Z 614.864,A -85,B 0,C 180,E1 15995.382,E2 15995.382} C_VEL
LIN {X 0,Y 308.853,Z 607.551,A -85,B 0,C 180,E1 15999.69,E2 15999.69} C_VEL
LIN {X 0,Y 302.714,Z 599.441,A -85,B 0,C 180,E1 16004.348,E2 16004.348} C_VEL
LIN {X 0,Y 299.169,Z 593.553,A -85,B 0,C 180,E1 16007.988,E2 16007.988} C_VEL
LIN {X 0,Y 295.537,Z 587.719,A -85,B 0,C 180,E1 16013.4,E2 16013.4} C_VEL
LIN {X 0,Y 294.437,Z 586.276,A -85,B 0,C 180,E1 16016.426,E2 16016.426} C_VEL
LIN {X 0,Y 295.539,Z 587.283,A -85,B 0,C 180,E1 16025.959,E2 16025.959} C_VEL
LIN {X 0,Y 299.119,Z 593.374,A -85,B 0,C 180,E1 16031.454,E2 16031.454} C_VEL
LIN {X 0,Y 300.746,Z 595.83,A -85,B 0,C 180,E1 16033.171,E2 16033.171} C_VEL
LIN {X 0,Y 305.53,Z 603.099,A -85,B 0,C 180,E1 16037.234,E2 16037.234} C_VEL
LIN {X 0,Y 312.897,Z 614.511,A -85,B 0,C 180,E1 16042.224,E2 16042.224} C_VEL
LIN {X 0,Y 324.006,Z 634.737,A -85,B 0,C 180,E1 16048.446,E2 16048.446} C_VEL
LIN {X 0,Y 333.494,Z 657.539,A -85,B 0,C 180,E1 16053.664,E2 16053.664} C_VEL
LIN {X 0,Y 340.176,Z 679.491,A -85,B 0,C 180,E1 16057.82,E2 16057.82} C_VEL
LIN {X 0,Y 329.223,Z 715.307,A -85,B 0,C 180,E1 16060.86,E2 16060.86} C_VEL
LIN {X 0,Y 317.07,Z 747.947,A -85,B 0,C 180,E1 16064.82,E2 16064.82} C_VEL
LIN {X 0,Y 303.975,Z 778.394,A -85,B 0,C 180,E1 16070.125,E2 16070.125} C_VEL
LIN {X 0,Y 292.682,Z 803.492,A -85,B 0,C 180,E1 16076.339,E2 16076.339} C_VEL
LIN {X 0,Y 283.629,Z 824.802,A -85,B 0,C 180,E1 16083.963,E2 16083.963} C_VEL
LIN {X 0,Y 278.518,Z 839.464,A -85,B 0,C 180,E1 16091.855,E2 16091.855} C_VEL
LIN {X 0,Y 276.578,Z 848.034,A -85,B 0,C 180,E1 16099.115,E2 16099.115} C_VEL
LIN {X 0,Y 276.056,Z 852.482,A -85,B 0,C 180,E1 16106.865,E2 16106.865} C_VEL
LIN {X 0,Y 276.069,Z 852.483,A -85,B 0,C 180,E1 16113.132,E2 16113.132} C_VEL
LIN {X 0,Y 276.544,Z 848.067,A -85,B 0,C 180,E1 16120.849,E2 16120.849} C_VEL
LIN {X 0,Y 278.939,Z 838.285,A -85,B 0,C 180,E1 16128.939,E2 16128.939} C_VEL
LIN {X 0,Y 284.441,Z 822.928,A -85,B 0,C 180,E1 16136.802,E2 16136.802} C_VEL
LIN {X 0,Y 293.267,Z 802.292,A -85,B 0,C 180,E1 16144.025,E2 16144.025} C_VEL
LIN {X 0,Y 305.187,Z 775.559,A -85,B 0,C 180,E1 16150.462,E2 16150.462} C_VEL
LIN {X 0,Y 317.677,Z 746.169,A -85,B 0,C 180,E1 16155.438,E2 16155.438} C_VEL
LIN {X 0,Y 330.742,Z 710.964,A -85,B 0,C 180,E1 16159.583,E2 16159.583} C_VEL
LIN {X 0,Y 340.205,Z 679.512,A -85,B 0,C 180,E1 16162.171,E2 16162.171} C_VEL
LIN {X 0,Y 332.365,Z 654.402,A -85,B 0,C 180,E1 16166.991,E2 16166.991} C_VEL
LIN {X 0,Y 322.517,Z 632.264,A -85,B 0,C 180,E1 16172.279,E2 16172.279} C_VEL
LIN {X 0,Y 322.332,Z 631.884,A -85,B 0,C 180,E1 16172.378,E2 16172.378} C_VEL
LIN {X 0,Y 317.498,Z 629.718,A -85,B 0,C 180,E1 16174.291,E2 16174.291} C_VEL
LIN {X 0,Y 313.535,Z 627.978,A -85,B 0,C 180,E1 16176.007,E2 16176.007} C_VEL
LIN {X 0,Y 313.188,Z 627.248,A -85,B 0,C 180,E1 16176.232,E2 16176.232} C_VEL
LIN {X 0,Y 305.055,Z 613.266,A -85,B 0,C 180,E1 16181.786,E2 16181.786} C_VEL
LIN {X 0,Y 301.062,Z 606.93,A -85,B 0,C 180,E1 16185.118,E2 16185.118} C_VEL
LIN {X 0,Y 297.606,Z 601.074,A -85,B 0,C 180,E1 16188.857,E2 16188.857} C_VEL
LIN {X 0,Y 294.234,Z 594.99,A -85,B 0,C 180,E1 16194.393,E2 16194.393} C_VEL
LIN {X 0,Y 293.371,Z 594.102,A -85,B 0,C 180,E1 16203.755,E2 16203.755} C_VEL
LIN {X 0,Y 294.334,Z 595.659,A -85,B 0,C 180,E1 16206.535,E2 16206.535} C_VEL
LIN {X 0,Y 298.705,Z 603.09,A -85,B 0,C 180,E1 16213.143,E2 16213.143} C_VEL
LIN {X 0,Y 303.546,Z 611.229,A -85,B 0,C 180,E1 16217.824,E2 16217.824} C_VEL
LIN {X 0,Y 309.607,Z 618.92,A -85,B 0,C 180,E1 16222.271,E2 16222.271} C_VEL
LIN {X 0,Y 316.723,Z 626.622,A -85,B 0,C 180,E1 16227.779,E2 16227.779} C_VEL
LIN {X 0,Y 322.838,Z 632.219,A -85,B 0,C 180,E1 16232.928,E2 16232.928} C_VEL
LIN {X 0,Y 329.029,Z 639.386,A -85,B 0,C 180,E1 16239.005,E2 16239.005} C_VEL
LIN {X 0,Y 332.222,Z 642.133,A -85,B 0,C 180,E1 16242.265,E2 16242.265} C_VEL
LIN {X 0,Y 337.17,Z 647.602,A -85,B 0,C 180,E1 16247.832,E2 16247.832} C_VEL
LIN {X 0,Y 340.508,Z 650.121,A -85,B 0,C 180,E1 16251.726,E2 16251.726} C_VEL
LIN {X 0,Y 344.501,Z 655.2,A -85,B 0,C 180,E1 16257.435,E2 16257.435} C_VEL
LIN {X 0,Y 348.691,Z 657.929,A -85,B 0,C 180,E1 16263.838,E2 16263.838} C_VEL
LIN {X 0,Y 351.507,Z 662.156,A -85,B 0,C 180,E1 16269.915,E2 16269.915} C_VEL
LIN {X 0,Y 354.063,Z 663.901,A -85,B 0,C 180,E1 16276.444,E2 16276.444} C_VEL
LIN {X 0,Y 355.579,Z 664.454,A -85,B 0,C 180,E1 16282.687,E2 16282.687} C_VEL
LIN {X 0,Y 356.182,Z 664.647,A -85,B 0,C 180,E1 16287.573,E2 16287.573} C_VEL
LIN {X 0,Y 355.958,Z 664.598,A -85,B 0,C 180,E1 16294.865,E2 16294.865} C_VEL
LIN {X 0,Y 354.546,Z 664.176,A -85,B 0,C 180,E1 16301.777,E2 16301.777} C_VEL
LIN {X 0,Y 352.161,Z 662.66,A -85,B 0,C 180,E1 16308.633,E2 16308.633} C_VEL
LIN {X 0,Y 349.259,Z 659.077,A -85,B 0,C 180,E1 16314.961,E2 16314.961} C_VEL
LIN {X 0,Y 347.845,Z 656.867,A -85,B 0,C 180,E1 16317.749,E2 16317.749} C_VEL
LIN {X 0,Y 343.165,Z 654.079,A -85,B 0,C 180,E1 16324.432,E2 16324.432} C_VEL
LIN {X 0,Y 339.013,Z 648.492,A -85,B 0,C 180,E1 16330.177,E2 16330.177} C_VEL
LIN {X 0,Y 333.803,Z 644.337,A -85,B 0,C 180,E1 16335.963,E2 16335.963} C_VEL
LIN {X 0,Y 330.692,Z 640.209,A -85,B 0,C 180,E1 16339.467,E2 16339.467} C_VEL
LIN {X 0,Y 325.172,Z 635.389,A -85,B 0,C 180,E1 16344.753,E2 16344.753} C_VEL
LIN {X 0,Y 322.094,Z 631.946,A -85,B 0,C 180,E1 16347.643,E2 16347.643} C_VEL
LIN {X 0,Y 316.032,Z 625.675,A -85,B 0,C 180,E1 16352.83,E2 16352.83} C_VEL
LIN {X 0,Y 309.06,Z 618.072,A -85,B 0,C 180,E1 16358.163,E2 16358.163} C_VEL
LIN {X 0,Y 300.184,Z 606.183,A -85,B 0,C 180,E1 16365.168,E2 16365.168} C_VEL
LIN {X 0,Y 297.328,Z 601.07,A -85,B 0,C 180,E1 16368.459,E2 16368.459} C_VEL
LIN {X 0,Y 294.188,Z 595.023,A -85,B 0,C 180,E1 16373.924,E2 16373.924} C_VEL
LIN {X 0,Y 293.278,Z 594.02,A -85,B 0,C 180,E1 16382.946,E2 16382.946} C_VEL
LIN {X 0,Y 294.311,Z 595.34,A -85,B 0,C 180,E1 16385.883,E2 16385.883} C_VEL
LIN {X 0,Y 298.128,Z 601.371,A -85,B 0,C 180,E1 16391.678,E2 16391.678} C_VEL
LIN {X 0,Y 303.584,Z 610.938,A -85,B 0,C 180,E1 16397.069,E2 16397.069} C_VEL
LIN {X 0,Y 310.163,Z 621.527,A -85,B 0,C 180,E1 16401.772,E2 16401.772} C_VEL
LIN {X 0,Y 319.781,Z 640.276,A -85,B 0,C 180,E1 16407.713,E2 16407.713} C_VEL
LIN {X 0,Y 328.554,Z 662.266,A -85,B 0,C 180,E1 16412.953,E2 16412.953} C_VEL
LIN {X 0,Y 334.27,Z 683.44,A -85,B 0,C 180,E1 16417.063,E2 16417.063} C_VEL
LIN {X 0,Y 321.396,Z 722.33,A -85,B 0,C 180,E1 16420.531,E2 16420.531} C_VEL
LIN {X 0,Y 307.751,Z 755.997,A -85,B 0,C 180,E1 16425.04,E2 16425.04} C_VEL
LIN {X 0,Y 294.961,Z 784.084,A -85,B 0,C 180,E1 16430.407,E2 16430.407} C_VEL
LIN {X 0,Y 283.181,Z 809.288,A -85,B 0,C 180,E1 16437.346,E2 16437.346} C_VEL
LIN {X 0,Y 274.531,Z 828.927,A -85,B 0,C 180,E1 16445.33,E2 16445.33} C_VEL
LIN {X 0,Y 270.333,Z 840.932,A -85,B 0,C 180,E1 16452.517,E2 16452.517} C_VEL
LIN {X 0,Y 268.516,Z 849.016,A -85,B 0,C 180,E1 16460.292,E2 16460.292} C_VEL
LIN {X 0,Y 268.148,Z 852.236,A -85,B 0,C 180,E1 16466.772,E2 16466.772} C_VEL
LIN {X 0,Y 268.159,Z 852.237,A -85,B 0,C 180,E1 16473.224,E2 16473.224} C_VEL
LIN {X 0,Y 268.675,Z 847.818,A -85,B 0,C 180,E1 16481.171,E2 16481.171} C_VEL
LIN {X 0,Y 271.26,Z 838.032,A -85,B 0,C 180,E1 16489.497,E2 16489.497} C_VEL
LIN {X 0,Y 277.16,Z 822.674,A -85,B 0,C 180,E1 16497.565,E2 16497.565} C_VEL
LIN {X 0,Y 286.542,Z 802.039,A -85,B 0,C 180,E1 16504.938,E2 16504.938} C_VEL
LIN {X 0,Y 299.068,Z 775.308,A -85,B 0,C 180,E1 16511.47,E2 16511.47} C_VEL
LIN {X 0,Y 312.049,Z 745.917,A -85,B 0,C 180,E1 16516.498,E2 16516.498} C_VEL
LIN {X 0,Y 325.606,Z 710.715,A -85,B 0,C 180,E1 16520.656,E2 16520.656} C_VEL
LIN {X 0,Y 334.319,Z 683.429,A -85,B 0,C 180,E1 16522.928,E2 16522.928} C_VEL
LIN {X 0,Y 328.572,Z 662.228,A -85,B 0,C 180,E1 16527.047,E2 16527.047} C_VEL
LIN {X 0,Y 320.394,Z 641.768,A -85,B 0,C 180,E1 16531.905,E2 16531.905} C_VEL
LIN {X 0,Y 313.188,Z 627.248,A -85,B 0,C 180,E1 16536.232,E2 16536.232} C_VEL
LIN {X 0,Y 309.462,Z 622.842,A -85,B 0,C 180,E1 16538.377,E2 16538.377} C_VEL
LIN {X 0,Y 302.454,Z 620.214,A -85,B 0,C 180,E1 16542.34,E2 16542.34} C_VEL
LIN {X 0,Y 298.478,Z 613.652,A -85,B 0,C 180,E1 16545.954,E2 16545.954} C_VEL
LIN {X 0,Y 295.608,Z 608.497,A -85,B 0,C 180,E1 16549.339,E2 16549.339} C_VEL
LIN {X 0,Y 292.483,Z 602.072,A -85,B 0,C 180,E1 16555.565,E2 16555.565} C_VEL
LIN {X 0,Y 292.687,Z 602.568,A -85,B 0,C 180,E1 16565.752,E2 16565.752} C_VEL
LIN {X 0,Y 295.785,Z 608.737,A -85,B 0,C 180,E1 16571.591,E2 16571.591} C_VEL
LIN {X 0,Y 301.036,Z 618.431,A -85,B 0,C 180,E1 16577.41,E2 16577.41} C_VEL
LIN {X 0,Y 307.492,Z 626.92,A -85,B 0,C 180,E1 16582.352,E2 16582.352} C_VEL
LIN {X 0,Y 314.187,Z 633.946,A -85,B 0,C 180,E1 16587.496,E2 16587.496} C_VEL
LIN {X 0,Y 320.633,Z 639.784,A -85,B 0,C 180,E1 16592.814,E2 16592.814} C_VEL
LIN {X 0,Y 326.983,Z 646.997,A -85,B 0,C 180,E1 16598.942,E2 16598.942} C_VEL
LIN {X 0,Y 330.343,Z 649.879,A -85,B 0,C 180,E1 16602.23,E2 16602.23} C_VEL
LIN {X 0,Y 335.677,Z 655.437,A -85,B 0,C 180,E1 16608.114,E2 16608.114} C_VEL
LIN {X 0,Y 338.647,Z 657.715,A -85,B 0,C 180,E1 16611.538,E2 16611.538} C_VEL
LIN {X 0,Y 342.995,Z 662.988,A -85,B 0,C 180,E1 16617.582,E2 16617.582} C_VEL
LIN {X 0,Y 347.231,Z 665.813,A -85,B 0,C 180,E1 16623.872,E2 16623.872} C_VEL
LIN {X 0,Y 350.151,Z 670.034,A -85,B 0,C 180,E1 16630.204,E2 16630.204} C_VEL
LIN {X 0,Y 352.628,Z 671.65,A -85,B 0,C 180,E1 16636.388,E2 16636.388} C_VEL
LIN {X 0,Y 354.231,Z 672.213,A -85,B 0,C 180,E1 16642.659,E2 16642.659} C_VEL
LIN {X 0,Y 354.863,Z 672.431,A -85,B 0,C 180,E1 16647.564,E2 16647.564} C_VEL
LIN {X 0,Y 354.626,Z 672.357,A -85,B 0,C 180,E1 16654.883,E2 16654.883} C_VEL
LIN {X 0,Y 353.243,Z 671.953,A -85,B 0,C 180,E1 16661.594,E2 16661.594} C_VEL
LIN {X 0,Y 350.751,Z 670.499,A -85,B 0,C 180,E1 16668.446,E2 16668.446} C_VEL
LIN {X 0,Y 347.747,Z 666.86,A -85,B 0,C 180,E1 16674.994,E2 16674.994} C_VEL
LIN {X 0,Y 346.001,Z 664.493,A -85,B 0,C 180,E1 16678.231,E2 16678.231} C_VEL
LIN {X 0,Y 341.095,Z 661.494,A -85,B 0,C 180,E1 16684.938,E2 16684.938} C_VEL
LIN {X 0,Y 337.036,Z 656.058,A -85,B 0,C 180,E1 16690.432,E2 16690.432} C_VEL
LIN {X 0,Y 331.644,Z 651.687,A -85,B 0,C 180,E1 16696.301,E2 16696.301} C_VEL
LIN {X 0,Y 328.264,Z 647.637,A -85,B 0,C 180,E1 16699.939,E2 16699.939} C_VEL
LIN {X 0,Y 322.475,Z 642.221,A -85,B 0,C 180,E1 16705.397,E2 16705.397} C_VEL
LIN {X 0,Y 318.978,Z 638.879,A -85,B 0,C 180,E1 16708.474,E2 16708.474} C_VEL
LIN {X 0,Y 313.149,Z 632.365,A -85,B 0,C 180,E1 16713.43,E2 16713.43} C_VEL
LIN {X 0,Y 306.452,Z 625.343,A -85,B 0,C 180,E1 16718.477,E2 16718.477} C_VEL
LIN {X 0,Y 297.622,Z 612.881,A -85,B 0,C 180,E1 16725.968,E2 16725.968} C_VEL
LIN {X 0,Y 295.337,Z 608.509,A -85,B 0,C 180,E1 16728.907,E2 16728.907} C_VEL
LIN {X 0,Y 292.473,Z 602.081,A -85,B 0,C 180,E1 16734.92,E2 16734.92} C_VEL
LIN {X 0,Y 292.792,Z 602.478,A -85,B 0,C 180,E1 16745.264,E2 16745.264} C_VEL
LIN {X 0,Y 296.097,Z 608.82,A -85,B 0,C 180,E1 16751.2,E2 16751.2} C_VEL
LIN {X 0,Y 301.385,Z 618.337,A -85,B 0,C 180,E1 16756.729,E2 16756.729} C_VEL
LIN {X 0,Y 307.64,Z 629.404,A -85,B 0,C 180,E1 16761.638,E2 16761.638} C_VEL
LIN {X 0,Y 316.211,Z 647.061,A -85,B 0,C 180,E1 16767.34,E2 16767.34} C_VEL
LIN {X 0,Y 323.849,Z 667.762,A -85,B 0,C 180,E1 16772.4,E2 16772.4} C_VEL
LIN {X 0,Y 328.498,Z 686.49,A -85,B 0,C 180,E1 16776.204,E2 16776.204} C_VEL
LIN {X 0,Y 315.681,Z 723.446,A -85,B 0,C 180,E1 16779.572,E2 16779.572} C_VEL
LIN {X 0,Y 301.338,Z 757.39,A -85,B 0,C 180,E1 16784.215,E2 16784.215} C_VEL
LIN {X 0,Y 287.682,Z 785.852,A -85,B 0,C 180,E1 16789.856,E2 16789.856} C_VEL
LIN {X 0,Y 275.767,Z 810.196,A -85,B 0,C 180,E1 16796.823,E2 16796.823} C_VEL
LIN {X 0,Y 267.058,Z 828.852,A -85,B 0,C 180,E1 16804.69,E2 16804.69} C_VEL
LIN {X 0,Y 262.14,Z 842.289,A -85,B 0,C 180,E1 16813.271,E2 16813.271} C_VEL
LIN {X 0,Y 260.467,Z 849.818,A -85,B 0,C 180,E1 16821.671,E2 16821.671} C_VEL
LIN {X 0,Y 260.417,Z 852.403,A -85,B 0,C 180,E1 16829.998,E2 16829.998} C_VEL
LIN {X 0,Y 260.445,Z 849.82,A -85,B 0,C 180,E1 16838.327,E2 16838.327} C_VEL
LIN {X 0,Y 262.164,Z 842.293,A -85,B 0,C 180,E1 16846.725,E2 16846.725} C_VEL
LIN {X 0,Y 266.347,Z 830.683,A -85,B 0,C 180,E1 16854.383,E2 16854.383} C_VEL
LIN {X 0,Y 275.12,Z 811.376,A -85,B 0,C 180,E1 16862.749,E2 16862.749} C_VEL
LIN {X 0,Y 286.768,Z 787.674,A -85,B 0,C 180,E1 16869.706,E2 16869.706} C_VEL
LIN {X 0,Y 300.648,Z 758.861,A -85,B 0,C 180,E1 16875.557,E2 16875.557} C_VEL
LIN {X 0,Y 315.209,Z 724.767,A -85,B 0,C 180,E1 16880.259,E2 16880.259} C_VEL
LIN {X 0,Y 327.131,Z 690.924,A -85,B 0,C 180,E1 16883.458,E2 16883.458} C_VEL
LIN {X 0,Y 328.512,Z 685.424,A -85,B 0,C 180,E1 16883.949,E2 16883.949} C_VEL
LIN {X 0,Y 321.862,Z 661.679,A -85,B 0,C 180,E1 16888.958,E2 16888.958} C_VEL
LIN {X 0,Y 312.845,Z 639.984,A -85,B 0,C 180,E1 16894.787,E2 16894.787} C_VEL
LIN {X 0,Y 303.786,Z 621.952,A -85,B 0,C 180,E1 16901.323,E2 16901.323} C_VEL
LIN {X 0,Y 302.454,Z 620.214,A -85,B 0,C 180,E1 16902.34,E2 16902.34} C_VEL
LIN {X 0,Y 294.368,Z 616.602,A -85,B 0,C 180,E1 16908.857,E2 16908.857} C_VEL
LIN {X 0,Y 291.087,Z 610.237,A -85,B 0,C 180,E1 16914.985,E2 16914.985} C_VEL
LIN {X 0,Y 290.71,Z 609.731,A -85,B 0,C 180,E1 16924.6,E2 16924.6} C_VEL
LIN {X 0,Y 294.572,Z 618.224,A -85,B 0,C 180,E1 16932.579,E2 16932.579} C_VEL
LIN {X 0,Y 304.399,Z 633.745,A -85,B 0,C 180,E1 16941.83,E2 16941.83} C_VEL
LIN {X 0,Y 311.014,Z 640.424,A -85,B 0,C 180,E1 16946.785,E2 16946.785} C_VEL
LIN {X 0,Y 317.69,Z 647.025,A -85,B 0,C 180,E1 16952.304,E2 16952.304} C_VEL
LIN {X 0,Y 324.707,Z 654.539,A -85,B 0,C 180,E1 16958.886,E2 16958.886} C_VEL
LIN {X 0,Y 328.049,Z 657.509,A -85,B 0,C 180,E1 16962.148,E2 16962.148} C_VEL
LIN {X 0,Y 333.329,Z 662.929,A -85,B 0,C 180,E1 16967.832,E2 16967.832} C_VEL
LIN {X 0,Y 336.637,Z 665.478,A -85,B 0,C 180,E1 16971.523,E2 16971.523} C_VEL
LIN {X 0,Y 341.154,Z 670.695,A -85,B 0,C 180,E1 16977.693,E2 16977.693} C_VEL
LIN {X 0,Y 345.321,Z 673.423,A -85,B 0,C 180,E1 16983.717,E2 16983.717} C_VEL
LIN {X 0,Y 348.318,Z 677.669,A -85,B 0,C 180,E1 16990.07,E2 16990.07} C_VEL
LIN {X 0,Y 350.899,Z 679.342,A -85,B 0,C 180,E1 16996.32,E2 16996.32} C_VEL
LIN {X 0,Y 352.6,Z 679.935,A -85,B 0,C 180,E1 17002.625,E2 17002.625} C_VEL
LIN {X 0,Y 353.25,Z 680.164,A -85,B 0,C 180,E1 17007.553,E2 17007.553} C_VEL
LIN {X 0,Y 353.001,Z 680.078,A -85,B 0,C 180,E1 17014.906,E2 17014.906} C_VEL
LIN {X 0,Y 351.571,Z 679.651,A -85,B 0,C 180,E1 17021.667,E2 17021.667} C_VEL
LIN {X 0,Y 348.949,Z 678.162,A -85,B 0,C 180,E1 17028.544,E2 17028.544} C_VEL
LIN {X 0,Y 345.862,Z 674.398,A -85,B 0,C 180,E1 17035.222,E2 17035.222} C_VEL
LIN {X 0,Y 343.877,Z 672.06,A -85,B 0,C 180,E1 17038.637,E2 17038.637} C_VEL
LIN {X 0,Y 338.808,Z 668.811,A -85,B 0,C 180,E1 17045.382,E2 17045.382} C_VEL
LIN {X 0,Y 335.072,Z 663.713,A -85,B 0,C 180,E1 17050.409,E2 17050.409} C_VEL
LIN {X 0,Y 329.419,Z 659.27,A -85,B 0,C 180,E1 17056.374,E2 17056.374} C_VEL
LIN {X 0,Y 326.406,Z 655.368,A -85,B 0,C 180,E1 17059.664,E2 17059.664} C_VEL
LIN {X 0,Y 320.386,Z 650.25,A -85,B 0,C 180,E1 17065.171,E2 17065.171} C_VEL
LIN {X 0,Y 318.564,Z 647.505,A -85,B 0,C 180,E1 17066.99,E2 17066.99} C_VEL
LIN {X 0,Y 311.724,Z 641.737,A -85,B 0,C 180,E1 17072.511,E2 17072.511} C_VEL
LIN {X 0,Y 308.075,Z 637.778,A -85,B 0,C 180,E1 17075.393,E2 17075.393} C_VEL
LIN {X 0,Y 297.853,Z 624.237,A -85,B 0,C 180,E1 17083.622,E2 17083.622} C_VEL
LIN {X 0,Y 293.208,Z 615.898,A -85,B 0,C 180,E1 17089.355,E2 17089.355} C_VEL
LIN {X 0,Y 290.601,Z 609.678,A -85,B 0,C 180,E1 17095.738,E2 17095.738} C_VEL
LIN {X 0,Y 291.132,Z 610.458,A -85,B 0,C 180,E1 17105.201,E2 17105.201} C_VEL
LIN {X 0,Y 295.079,Z 618.397,A -85,B 0,C 180,E1 17112.182,E2 17112.182} C_VEL
LIN {X 0,Y 299.598,Z 626.957,A -85,B 0,C 180,E1 17117.068,E2 17117.068} C_VEL
LIN {X 0,Y 306.667,Z 640.571,A -85,B 0,C 180,E1 17122.796,E2 17122.796} C_VEL
LIN {X 0,Y 315.19,Z 660.997,A -85,B 0,C 180,E1 17128.926,E2 17128.926} C_VEL
LIN {X 0,Y 322.209,Z 685.824,A -85,B 0,C 180,E1 17134.597,E2 17134.597} C_VEL
LIN {X 0,Y 322.284,Z 691.107,A -85,B 0,C 180,E1 17135.43,E2 17135.43} C_VEL
LIN {X 0,Y 309.496,Z 725.79,A -85,B 0,C 180,E1 17138.727,E2 17138.727} C_VEL
LIN {X 0,Y 294.631,Z 759.562,A -85,B 0,C 180,E1 17143.483,E2 17143.483} C_VEL
LIN {X 0,Y 279.698,Z 789.12,A -85,B 0,C 180,E1 17149.651,E2 17149.651} C_VEL
LIN {X 0,Y 267.933,Z 811.846,A -85,B 0,C 180,E1 17156.583,E2 17156.583} C_VEL
LIN {X 0,Y 258.932,Z 830.452,A -85,B 0,C 180,E1 17164.884,E2 17164.884} C_VEL
LIN {X 0,Y 254.404,Z 842.038,A -85,B 0,C 180,E1 17172.746,E2 17172.746} C_VEL
LIN {X 0,Y 252.607,Z 849.611,A -85,B 0,C 180,E1 17181.475,E2 17181.475} C_VEL
LIN {X 0,Y 252.515,Z 852.158,A -85,B 0,C 180,E1 17189.998,E2 17189.998} C_VEL
LIN {X 0,Y 252.583,Z 849.623,A -85,B 0,C 180,E1 17198.506,E2 17198.506} C_VEL
LIN {X 0,Y 254.436,Z 842.042,A -85,B 0,C 180,E1 17207.248,E2 17207.248} C_VEL
LIN {X 0,Y 258.949,Z 830.43,A -85,B 0,C 180,E1 17215.127,E2 17215.127} C_VEL
LIN {X 0,Y 267.887,Z 811.875,A -85,B 0,C 180,E1 17223.41,E2 17223.41} C_VEL
LIN {X 0,Y 279.685,Z 789.131,A -85,B 0,C 180,E1 17230.347,E2 17230.347} C_VEL
LIN {X 0,Y 294.525,Z 759.697,A -85,B 0,C 180,E1 17236.502,E2 17236.502} C_VEL
LIN {X 0,Y 309.57,Z 725.814,A -85,B 0,C 180,E1 17241.252,E2 17241.252} C_VEL
LIN {X 0,Y 321.944,Z 692.207,A -85,B 0,C 180,E1 17244.484,E2 17244.484} C_VEL
LIN {X 0,Y 322.58,Z 687.57,A -85,B 0,C 180,E1 17245.041,E2 17245.041} C_VEL
LIN {X 0,Y 316.399,Z 664.453,A -85,B 0,C 180,E1 17250.218,E2 17250.218} C_VEL
LIN {X 0,Y 308.027,Z 643.731,A -85,B 0,C 180,E1 17256.165,E2 17256.165} C_VEL
LIN {X 0,Y 300.393,Z 628.133,A -85,B 0,C 180,E1 17262.268,E2 17262.268} C_VEL
LIN {X 0,Y 295.647,Z 619.981,A -85,B 0,C 180,E1 17266.995,E2 17266.995} C_VEL
LIN {X 0,Y 294.368,Z 616.602,A -85,B 0,C 180,E1 17268.857,E2 17268.857} C_VEL
LIN {X 0,Y 291.45,Z 616.347,A -85,B 0,C 180,E1 17272.196,E2 17272.196} C_VEL
LIN {X 0,Y 289.188,Z 617.524,A -85,B 0,C 180,E1 17275.619,E2 17275.619} C_VEL
LIN {X 0,Y 289.123,Z 617.887,A -85,B 0,C 180,E1 17285.31,E2 17285.31} C_VEL
LIN {X 0,Y 292.372,Z 625.946,A -85,B 0,C 180,E1 17292.485,E2 17292.485} C_VEL
LIN {X 0,Y 303.804,Z 643.792,A -85,B 0,C 180,E1 17303.416,E2 17303.416} C_VEL
LIN {X 0,Y 309.443,Z 649.572,A -85,B 0,C 180,E1 17307.735,E2 17307.735} C_VEL
LIN {X 0,Y 317.142,Z 656.638,A -85,B 0,C 180,E1 17314.069,E2 17314.069} C_VEL
LIN {X 0,Y 320.907,Z 661.096,A -85,B 0,C 180,E1 17317.687,E2 17317.687} C_VEL
LIN {X 0,Y 324.886,Z 663.931,A -85,B 0,C 180,E1 17321.299,E2 17321.299} C_VEL
LIN {X 0,Y 330.204,Z 669.975,A -85,B 0,C 180,E1 17326.989,E2 17326.989} C_VEL
LIN {X 0,Y 334.277,Z 672.952,A -85,B 0,C 180,E1 17331.385,E2 17331.385} C_VEL
LIN {X 0,Y 339.028,Z 678.301,A -85,B 0,C 180,E1 17337.749,E2 17337.749} C_VEL
LIN {X 0,Y 343.12,Z 680.923,A -85,B 0,C 180,E1 17343.535,E2 17343.535} C_VEL
LIN {X 0,Y 346.21,Z 685.246,A -85,B 0,C 180,E1 17349.927,E2 17349.927} C_VEL
LIN {X 0,Y 348.784,Z 686.948,A -85,B 0,C 180,E1 17356,E2 17356} C_VEL
LIN {X 0,Y 350.673,Z 687.596,A -85,B 0,C 180,E1 17362.584,E2 17362.584} C_VEL
LIN {X 0,Y 351.349,Z 687.8,A -85,B 0,C 180,E1 17367.54,E2 17367.54} C_VEL
LIN {X 0,Y 351.329,Z 687.751,A -85,B 0,C 180,E1 17372.463,E2 17372.463} C_VEL
LIN {X 0,Y 350.526,Z 687.665,A -85,B 0,C 180,E1 17378.037,E2 17378.037} C_VEL
LIN {X 0,Y 348.61,Z 686.833,A -85,B 0,C 180,E1 17384.454,E2 17384.454} C_VEL
LIN {X 0,Y 345.764,Z 684.713,A -85,B 0,C 180,E1 17391.053,E2 17391.053} C_VEL
LIN {X 0,Y 342.689,Z 679.923,A -85,B 0,C 180,E1 17397.43,E2 17397.43} C_VEL
LIN {X 0,Y 337.594,Z 677.322,A -85,B 0,C 180,E1 17404.076,E2 17404.076} C_VEL
LIN {X 0,Y 333.499,Z 671.55,A -85,B 0,C 180,E1 17409.714,E2 17409.714} C_VEL
LIN {X 0,Y 328.605,Z 668.65,A -85,B 0,C 180,E1 17414.663,E2 17414.663} C_VEL
LIN {X 0,Y 324.354,Z 663.089,A -85,B 0,C 180,E1 17419.355,E2 17419.355} C_VEL
LIN {X 0,Y 317.772,Z 657.692,A -85,B 0,C 180,E1 17425.258,E2 17425.258} C_VEL
LIN {X 0,Y 312.69,Z 653.018,A -85,B 0,C 180,E1 17429.55,E2 17429.55} C_VEL
LIN {X 0,Y 306.072,Z 645.606,A -85,B 0,C 180,E1 17435.001,E2 17435.001} C_VEL
LIN {X 0,Y 300.204,Z 638.993,A -85,B 0,C 180,E1 17439.396,E2 17439.396} C_VEL
LIN {X 0,Y 291.121,Z 623.505,A -85,B 0,C 180,E1 17449.456,E2 17449.456} C_VEL
LIN {X 0,Y 288.863,Z 617.371,A -85,B 0,C 180,E1 17455.712,E2 17455.712} C_VEL
LIN {X 0,Y 289.313,Z 618.076,A -85,B 0,C 180,E1 17464.953,E2 17464.953} C_VEL
LIN {X 0,Y 292.767,Z 625.837,A -85,B 0,C 180,E1 17471.895,E2 17471.895} C_VEL
LIN {X 0,Y 298.052,Z 635.799,A -85,B 0,C 180,E1 17477.681,E2 17477.681} C_VEL
LIN {X 0,Y 305.804,Z 653.346,A -85,B 0,C 180,E1 17484.407,E2 17484.407} C_VEL
LIN {X 0,Y 312.683,Z 672.972,A -85,B 0,C 180,E1 17489.965,E2 17489.965} C_VEL
LIN {X 0,Y 317.083,Z 691.751,A -85,B 0,C 180,E1 17494.235,E2 17494.235} C_VEL
LIN {X 0,Y 303.943,Z 726.856,A -85,B 0,C 180,E1 17497.698,E2 17497.698} C_VEL
LIN {X 0,Y 288.779,Z 759.95,A -85,B 0,C 180,E1 17502.428,E2 17502.428} C_VEL
LIN {X 0,Y 273.506,Z 788.866,A -85,B 0,C 180,E1 17508.54,E2 17508.54} C_VEL
LIN {X 0,Y 260.981,Z 811.831,A -85,B 0,C 180,E1 17515.682,E2 17515.682} C_VEL
LIN {X 0,Y 251.511,Z 830.292,A -85,B 0,C 180,E1 17524.143,E2 17524.143} C_VEL
LIN {X 0,Y 246.696,Z 841.787,A -85,B 0,C 180,E1 17532.189,E2 17532.189} C_VEL
LIN {X 0,Y 244.78,Z 848.951,A -85,B 0,C 180,E1 17540.498,E2 17540.498} C_VEL
LIN {X 0,Y 244.44,Z 851.498,A -85,B 0,C 180,E1 17546.459,E2 17546.459} C_VEL
LIN {X 0,Y 244.447,Z 851.499,A -85,B 0,C 180,E1 17553.538,E2 17553.538} C_VEL
LIN {X 0,Y 245.179,Z 846.924,A -85,B 0,C 180,E1 17562.438,E2 17562.438} C_VEL
LIN {X 0,Y 248.414,Z 837.275,A -85,B 0,C 180,E1 17571.373,E2 17571.373} C_VEL
LIN {X 0,Y 255.649,Z 821.912,A -85,B 0,C 180,E1 17580.112,E2 17580.112} C_VEL
LIN {X 0,Y 266.885,Z 801.102,A -85,B 0,C 180,E1 17588.016,E2 17588.016} C_VEL
LIN {X 0,Y 281.086,Z 774.839,A -85,B 0,C 180,E1 17594.703,E2 17594.703} C_VEL
LIN {X 0,Y 295.863,Z 745.163,A -85,B 0,C 180,E1 17599.91,E2 17599.91} C_VEL
LIN {X 0,Y 310.914,Z 709.777,A -85,B 0,C 180,E1 17604.124,E2 17604.124} C_VEL
LIN {X 0,Y 317.11,Z 691.683,A -85,B 0,C 180,E1 17605.769,E2 17605.769} C_VEL
LIN {X 0,Y 311.223,Z 668.157,A -85,B 0,C 180,E1 17611.278,E2 17611.278} C_VEL
LIN {X 0,Y 303.204,Z 647.276,A -85,B 0,C 180,E1 17617.702,E2 17617.702} C_VEL
LIN {X 0,Y 296.668,Z 633.676,A -85,B 0,C 180,E1 17623.569,E2 17623.569} C_VEL
LIN {X 0,Y 291.901,Z 623.858,A -85,B 0,C 180,E1 17629.428,E2 17629.428} C_VEL
LIN {X 0,Y 289.188,Z 617.524,A -85,B 0,C 180,E1 17635.619,E2 17635.619} C_VEL
LIN {X 0,Y 287.374,Z 620.937,A -85,B 0,C 180,E1 17639.022,E2 17639.022} C_VEL
LIN {X 0,Y 286.463,Z 624.749,A -85,B 0,C 180,E1 17642.456,E2 17642.456} C_VEL
LIN {X 0,Y 287.051,Z 626.268,A -85,B 0,C 180,E1 17645.607,E2 17645.607} C_VEL
LIN {X 0,Y 289.779,Z 633.166,A -85,B 0,C 180,E1 17652.121,E2 17652.121} C_VEL
LIN {X 0,Y 301.3,Z 651.453,A -85,B 0,C 180,E1 17663.623,E2 17663.623} C_VEL
LIN {X 0,Y 308.476,Z 659.037,A -85,B 0,C 180,E1 17669.29,E2 17669.29} C_VEL
LIN {X 0,Y 314.652,Z 664.627,A -85,B 0,C 180,E1 17674.376,E2 17674.376} C_VEL
LIN {X 0,Y 322.391,Z 671.816,A -85,B 0,C 180,E1 17681.506,E2 17681.506} C_VEL
LIN {X 0,Y 328.029,Z 677.643,A -85,B 0,C 180,E1 17687.398,E2 17687.398} C_VEL
LIN {X 0,Y 331.309,Z 679.706,A -85,B 0,C 180,E1 17690.745,E2 17690.745} C_VEL
LIN {X 0,Y 335.198,Z 684.818,A -85,B 0,C 180,E1 17695.982,E2 17695.982} C_VEL
LIN {X 0,Y 340.266,Z 687.459,A -85,B 0,C 180,E1 17702.497,E2 17702.497} C_VEL
LIN {X 0,Y 342.76,Z 691.636,A -85,B 0,C 180,E1 17707.602,E2 17707.602} C_VEL
LIN {X 0,Y 346.072,Z 694.278,A -85,B 0,C 180,E1 17714.835,E2 17714.835} C_VEL
LIN {X 0,Y 347.817,Z 694.983,A -85,B 0,C 180,E1 17720.007,E2 17720.007} C_VEL
LIN {X 0,Y 348.907,Z 695.361,A -85,B 0,C 180,E1 17725.039,E2 17725.039} C_VEL
LIN {X 0,Y 349.209,Z 695.402,A -85,B 0,C 180,E1 17730.001,E2 17730.001} C_VEL
LIN {X 0,Y 348.803,Z 695.308,A -85,B 0,C 180,E1 17735.693,E2 17735.693} C_VEL
LIN {X 0,Y 347.04,Z 694.691,A -85,B 0,C 180,E1 17742.558,E2 17742.558} C_VEL
LIN {X 0,Y 344.916,Z 693.57,A -85,B 0,C 180,E1 17747.835,E2 17747.835} C_VEL
LIN {X 0,Y 342.256,Z 691.007,A -85,B 0,C 180,E1 17753.38,E2 17753.38} C_VEL
LIN {X 0,Y 340.272,Z 687.418,A -85,B 0,C 180,E1 17757.504,E2 17757.504} C_VEL
LIN {X 0,Y 336.288,Z 685.761,A -85,B 0,C 180,E1 17762.581,E2 17762.581} C_VEL
LIN {X 0,Y 332.313,Z 681.763,A -85,B 0,C 180,E1 17767.705,E2 17767.705} C_VEL
LIN {X 0,Y 331.019,Z 679.27,A -85,B 0,C 180,E1 17769.66,E2 17769.66} C_VEL
LIN {X 0,Y 324.89,Z 674.941,A -85,B 0,C 180,E1 17775.834,E2 17775.834} C_VEL
LIN {X 0,Y 320.128,Z 669.642,A -85,B 0,C 180,E1 17780.704,E2 17780.704} C_VEL
LIN {X 0,Y 314.591,Z 664.638,A -85,B 0,C 180,E1 17785.65,E2 17785.65} C_VEL
LIN {X 0,Y 306.215,Z 656.813,A -85,B 0,C 180,E1 17792.505,E2 17792.505} C_VEL
LIN {X 0,Y 297.564,Z 647.051,A -85,B 0,C 180,E1 17799.205,E2 17799.205} C_VEL
LIN {X 0,Y 288.758,Z 630.981,A -85,B 0,C 180,E1 17809.648,E2 17809.648} C_VEL
LIN {X 0,Y 286.879,Z 624.987,A -85,B 0,C 180,E1 17815.682,E2 17815.682} C_VEL
LIN {X 0,Y 287.228,Z 625.749,A -85,B 0,C 180,E1 17824.8,E2 17824.8} C_VEL
LIN {X 0,Y 290.476,Z 633.578,A -85,B 0,C 180,E1 17831.792,E2 17831.792} C_VEL
LIN {X 0,Y 295.509,Z 644.135,A -85,B 0,C 180,E1 17837.838,E2 17837.838} C_VEL
LIN {X 0,Y 302.349,Z 660.76,A -85,B 0,C 180,E1 17844.268,E2 17844.268} C_VEL
LIN {X 0,Y 308.54,Z 680.67,A -85,B 0,C 180,E1 17849.928,E2 17849.928} C_VEL
LIN {X 0,Y 311.508,Z 694.946,A -85,B 0,C 180,E1 17853.294,E2 17853.294} C_VEL
LIN {X 0,Y 296.863,Z 731.756,A -85,B 0,C 180,E1 17857.107,E2 17857.107} C_VEL
LIN {X 0,Y 281.7,Z 762.771,A -85,B 0,C 180,E1 17861.78,E2 17861.78} C_VEL
LIN {X 0,Y 265.821,Z 791.588,A -85,B 0,C 180,E1 17868.16,E2 17868.16} C_VEL
LIN {X 0,Y 251.928,Z 815.867,A -85,B 0,C 180,E1 17876.352,E2 17876.352} C_VEL
LIN {X 0,Y 242.726,Z 833.008,A -85,B 0,C 180,E1 17885.186,E2 17885.186} C_VEL
LIN {X 0,Y 238.325,Z 843.445,A -85,B 0,C 180,E1 17893.444,E2 17893.444} C_VEL
LIN {X 0,Y 236.684,Z 850.038,A -85,B 0,C 180,E1 17902.672,E2 17902.672} C_VEL
LIN {X 0,Y 236.734,Z 851.668,A -85,B 0,C 180,E1 17909.998,E2 17909.998} C_VEL
LIN {X 0,Y 236.667,Z 850.039,A -85,B 0,C 180,E1 17917.325,E2 17917.325} C_VEL
LIN {X 0,Y 238.356,Z 843.45,A -85,B 0,C 180,E1 17926.551,E2 17926.551} C_VEL
LIN {X 0,Y 243.415,Z 831.61,A -85,B 0,C 180,E1 17935.717,E2 17935.717} C_VEL
LIN {X 0,Y 252.447,Z 814.801,A -85,B 0,C 180,E1 17944.081,E2 17944.081} C_VEL
LIN {X 0,Y 265.799,Z 791.597,A -85,B 0,C 180,E1 17951.84,E2 17951.84} C_VEL
LIN {X 0,Y 281.596,Z 762.877,A -85,B 0,C 180,E1 17958.211,E2 17958.211} C_VEL
LIN {X 0,Y 296.503,Z 732.656,A -85,B 0,C 180,E1 17962.776,E2 17962.776} C_VEL
LIN {X 0,Y 310.985,Z 697.126,A -85,B 0,C 180,E1 17966.437,E2 17966.437} C_VEL
LIN {X 0,Y 310.954,Z 691.929,A -85,B 0,C 180,E1 17967.372,E2 17967.372} C_VEL
LIN {X 0,Y 305.719,Z 670.838,A -85,B 0,C 180,E1 17972.679,E2 17972.679} C_VEL
LIN {X 0,Y 299.245,Z 652.68,A -85,B 0,C 180,E1 17978.559,E2 17978.559} C_VEL
LIN {X 0,Y 292.301,Z 637.086,A -85,B 0,C 180,E1 17985.809,E2 17985.809} C_VEL
LIN {X 0,Y 288.958,Z 630.71,A -85,B 0,C 180,E1 17990.611,E2 17990.611} C_VEL
LIN {X 0,Y 286.979,Z 625.063,A -85,B 0,C 180,E1 17996.235,E2 17996.235} C_VEL
LIN {X 0,Y 286.463,Z 624.749,A -85,B 0,C 180,E1 18002.456,E2 18002.456} C_VEL
LIN {X 0,Y 286.178,Z 628.356,A -85,B 0,C 180,E1 18004.964,E2 18004.964} C_VEL
LIN {X 0,Y 285.529,Z 636.987,A -85,B 0,C 180,E1 18008.595,E2 18008.595} C_VEL
LIN {X 0,Y 285.69,Z 637.459,A -85,B 0,C 180,E1 18009.03,E2 18009.03} C_VEL
LIN {X 0,Y 288.66,Z 644.034,A -85,B 0,C 180,E1 18014.381,E2 18014.381} C_VEL
LIN {X 0,Y 298.52,Z 659.028,A -85,B 0,C 180,E1 18023.856,E2 18023.856} C_VEL
LIN {X 0,Y 307.644,Z 668.141,A -85,B 0,C 180,E1 18031.002,E2 18031.002} C_VEL
LIN {X 0,Y 314.271,Z 675.057,A -85,B 0,C 180,E1 18036.887,E2 18036.887} C_VEL
LIN {X 0,Y 319.432,Z 679.123,A -85,B 0,C 180,E1 18041.407,E2 18041.407} C_VEL
LIN {X 0,Y 325.665,Z 685.279,A -85,B 0,C 180,E1 18047.852,E2 18047.852} C_VEL
LIN {X 0,Y 328.85,Z 687.843,A -85,B 0,C 180,E1 18051.272,E2 18051.272} C_VEL
LIN {X 0,Y 333.293,Z 692.886,A -85,B 0,C 180,E1 18057.092,E2 18057.092} C_VEL
LIN {X 0,Y 338.084,Z 695.987,A -85,B 0,C 180,E1 18063.492,E2 18063.492} C_VEL
LIN {X 0,Y 340.976,Z 699.908,A -85,B 0,C 180,E1 18069.266,E2 18069.266} C_VEL
LIN {X 0,Y 343.575,Z 701.791,A -85,B 0,C 180,E1 18075.08,E2 18075.08} C_VEL
LIN {X 0,Y 345.274,Z 702.455,A -85,B 0,C 180,E1 18079.933,E2 18079.933} C_VEL
LIN {X 0,Y 346.401,Z 702.851,A -85,B 0,C 180,E1 18085.003,E2 18085.003} C_VEL
LIN {X 0,Y 346.726,Z 702.888,A -85,B 0,C 180,E1 18090.001,E2 18090.001} C_VEL
LIN {X 0,Y 346.363,Z 702.791,A -85,B 0,C 180,E1 18095,E2 18095} C_VEL
LIN {X 0,Y 345.3,Z 702.554,A -85,B 0,C 180,E1 18100.069,E2 18100.069} C_VEL
LIN {X 0,Y 343.405,Z 701.69,A -85,B 0,C 180,E1 18105.288,E2 18105.288} C_VEL
LIN {X 0,Y 340.577,Z 699.536,A -85,B 0,C 180,E1 18111.489,E2 18111.489} C_VEL
LIN {X 0,Y 338.01,Z 695.707,A -85,B 0,C 180,E1 18116.758,E2 18116.758} C_VEL
LIN {X 0,Y 333.295,Z 692.97,A -85,B 0,C 180,E1 18122.91,E2 18122.91} C_VEL
LIN {X 0,Y 328.821,Z 688.017,A -85,B 0,C 180,E1 18128.722,E2 18128.722} C_VEL
LIN {X 0,Y 323.388,Z 683.651,A -85,B 0,C 180,E1 18134.424,E2 18134.424} C_VEL
LIN {X 0,Y 318.905,Z 678.195,A -85,B 0,C 180,E1 18139.211,E2 18139.211} C_VEL
LIN {X 0,Y 311.861,Z 672.477,A -85,B 0,C 180,E1 18145.347,E2 18145.347} C_VEL
LIN {X 0,Y 307.611,Z 668.209,A -85,B 0,C 180,E1 18148.994,E2 18148.994} C_VEL
LIN {X 0,Y 298.561,Z 659.041,A -85,B 0,C 180,E1 18156.147,E2 18156.147} C_VEL
LIN {X 0,Y 286.582,Z 638.714,A -85,B 0,C 180,E1 18169.377,E2 18169.377} C_VEL
LIN {X 0,Y 284.542,Z 632.516,A -85,B 0,C 180,E1 18176.196,E2 18176.196} C_VEL
LIN {X 0,Y 284.997,Z 633.373,A -85,B 0,C 180,E1 18184.647,E2 18184.647} C_VEL
LIN {X 0,Y 287.721,Z 640.62,A -85,B 0,C 180,E1 18191.339,E2 18191.339} C_VEL
LIN {X 0,Y 292.799,Z 652.329,A -85,B 0,C 180,E1 18198.009,E2 18198.009} C_VEL
LIN {X 0,Y 298.913,Z 668.808,A -85,B 0,C 180,E1 18204.367,E2 18204.367} C_VEL
LIN {X 0,Y 303.918,Z 687.606,A -85,B 0,C 180,E1 18209.766,E2 18209.766} C_VEL
LIN {X 0,Y 305.675,Z 699.337,A -85,B 0,C 180,E1 18212.528,E2 18212.528} C_VEL
LIN {X 0,Y 290.707,Z 734.519,A -85,B 0,C 180,E1 18216.212,E2 18216.212} C_VEL
LIN {X 0,Y 273.724,Z 767.278,A -85,B 0,C 180,E1 18221.413,E2 18221.413} C_VEL
LIN {X 0,Y 258.941,Z 792.691,A -85,B 0,C 180,E1 18227.352,E2 18227.352} C_VEL
LIN {X 0,Y 244.547,Z 816.673,A -85,B 0,C 180,E1 18235.73,E2 18235.73} C_VEL
LIN {X 0,Y 234.597,Z 834.225,A -85,B 0,C 180,E1 18245.332,E2 18245.332} C_VEL
LIN {X 0,Y 229.982,Z 844.944,A -85,B 0,C 180,E1 18254.782,E2 18254.782} C_VEL
LIN {X 0,Y 228.789,Z 849.791,A -85,B 0,C 180,E1 18262.418,E2 18262.418} C_VEL
LIN {X 0,Y 228.831,Z 851.422,A -85,B 0,C 180,E1 18269.998,E2 18269.998} C_VEL
LIN {X 0,Y 228.821,Z 849.393,A -85,B 0,C 180,E1 18278.459,E2 18278.459} C_VEL
LIN {X 0,Y 230.615,Z 843.198,A -85,B 0,C 180,E1 18287.123,E2 18287.123} C_VEL
LIN {X 0,Y 236.091,Z 831.357,A -85,B 0,C 180,E1 18296.576,E2 18296.576} C_VEL
LIN {X 0,Y 245.69,Z 814.546,A -85,B 0,C 180,E1 18305.154,E2 18305.154} C_VEL
LIN {X 0,Y 259.749,Z 791.343,A -85,B 0,C 180,E1 18313.046,E2 18313.046} C_VEL
LIN {X 0,Y 276.422,Z 762.361,A -85,B 0,C 180,E1 18319.51,E2 18319.51} C_VEL
LIN {X 0,Y 291.666,Z 732.452,A -85,B 0,C 180,E1 18324.034,E2 18324.034} C_VEL
LIN {X 0,Y 305.843,Z 698.058,A -85,B 0,C 180,E1 18327.675,E2 18327.675} C_VEL
LIN {X 0,Y 301.282,Z 676.722,A -85,B 0,C 180,E1 18333.21,E2 18333.21} C_VEL
LIN {X 0,Y 295.096,Z 658.14,A -85,B 0,C 180,E1 18339.49,E2 18339.49} C_VEL
LIN {X 0,Y 289.238,Z 643.913,A -85,B 0,C 180,E1 18346.425,E2 18346.425} C_VEL
LIN {X 0,Y 286.41,Z 638.073,A -85,B 0,C 180,E1 18350.909,E2 18350.909} C_VEL
LIN {X 0,Y 284.65,Z 632.478,A -85,B 0,C 180,E1 18356.964,E2 18356.964} C_VEL
LIN {X 0,Y 284.725,Z 633.291,A -85,B 0,C 180,E1 18365.039,E2 18365.039} C_VEL
LIN {X 0,Y 285.69,Z 637.459,A -85,B 0,C 180,E1 18369.03,E2 18369.03} C_VEL
LIN {X 0,Y 285.592,Z 641.498,A -85,B 0,C 180,E1 18370.597,E2 18370.597} C_VEL
LIN {X 0,Y 284.865,Z 649.453,A -85,B 0,C 180,E1 18372.791,E2 18372.791} C_VEL
LIN {X 0,Y 284.989,Z 649.922,A -85,B 0,C 180,E1 18373.075,E2 18373.075} C_VEL
LIN {X 0,Y 296.721,Z 667.497,A -85,B 0,C 180,E1 18384.897,E2 18384.897} C_VEL
LIN {X 0,Y 304.811,Z 675.625,A -85,B 0,C 180,E1 18391.323,E2 18391.323} C_VEL
LIN {X 0,Y 313.311,Z 683.877,A -85,B 0,C 180,E1 18398.768,E2 18398.768} C_VEL
LIN {X 0,Y 319.565,Z 690.391,A -85,B 0,C 180,E1 18404.904,E2 18404.904} C_VEL
LIN {X 0,Y 325.159,Z 694.279,A -85,B 0,C 180,E1 18410.432,E2 18410.432} C_VEL
LIN {X 0,Y 329.987,Z 699.965,A -85,B 0,C 180,E1 18416.72,E2 18416.72} C_VEL
LIN {X 0,Y 332.834,Z 701.505,A -85,B 0,C 180,E1 18420.086,E2 18420.086} C_VEL
LIN {X 0,Y 335.473,Z 703.895,A -85,B 0,C 180,E1 18424.114,E2 18424.114} C_VEL
LIN {X 0,Y 338.222,Z 707.355,A -85,B 0,C 180,E1 18429.548,E2 18429.548} C_VEL
LIN {X 0,Y 341.323,Z 709.396,A -85,B 0,C 180,E1 18436.572,E2 18436.572} C_VEL
LIN {X 0,Y 343.147,Z 710.032,A -85,B 0,C 180,E1 18442.42,E2 18442.42} C_VEL
LIN {X 0,Y 343.873,Z 710.271,A -85,B 0,C 180,E1 18447.486,E2 18447.486} C_VEL
LIN {X 0,Y 343.865,Z 710.221,A -85,B 0,C 180,E1 18452.516,E2 18452.516} C_VEL
LIN {X 0,Y 343.091,Z 710.09,A -85,B 0,C 180,E1 18457.583,E2 18457.583} C_VEL
LIN {X 0,Y 341.309,Z 709.403,A -85,B 0,C 180,E1 18463.418,E2 18463.418} C_VEL
LIN {X 0,Y 337.988,Z 707.154,A -85,B 0,C 180,E1 18470.928,E2 18470.928} C_VEL
LIN {X 0,Y 335.012,Z 703.086,A -85,B 0,C 180,E1 18476.773,E2 18476.773} C_VEL
LIN {X 0,Y 329.981,Z 700.02,A -85,B 0,C 180,E1 18483.284,E2 18483.284} C_VEL
LIN {X 0,Y 325.126,Z 694.39,A -85,B 0,C 180,E1 18489.582,E2 18489.582} C_VEL
LIN {X 0,Y 318.257,Z 688.9,A -85,B 0,C 180,E1 18496.468,E2 18496.468} C_VEL
LIN {X 0,Y 313.38,Z 683.871,A -85,B 0,C 180,E1 18501.243,E2 18501.243} C_VEL
LIN {X 0,Y 306.634,Z 677.19,A -85,B 0,C 180,E1 18507.223,E2 18507.223} C_VEL
LIN {X 0,Y 298.412,Z 669.591,A -85,B 0,C 180,E1 18513.691,E2 18513.691} C_VEL
LIN {X 0,Y 286.736,Z 654.618,A -85,B 0,C 180,E1 18523.958,E2 18523.958} C_VEL
LIN {X 0,Y 283.158,Z 645.166,A -85,B 0,C 180,E1 18530.797,E2 18530.797} C_VEL
LIN {X 0,Y 282.046,Z 639.93,A -85,B 0,C 180,E1 18536.93,E2 18536.93} C_VEL
LIN {X 0,Y 282.302,Z 640.025,A -85,B 0,C 180,E1 18543.061,E2 18543.061} C_VEL
LIN {X 0,Y 285.157,Z 648.484,A -85,B 0,C 180,E1 18551.443,E2 18551.443} C_VEL
LIN {X 0,Y 289.89,Z 660.37,A -85,B 0,C 180,E1 18558.196,E2 18558.196} C_VEL
LIN {X 0,Y 295.432,Z 677.439,A -85,B 0,C 180,E1 18564.674,E2 18564.674} C_VEL
LIN {X 0,Y 299.61,Z 696.979,A -85,B 0,C 180,E1 18570.238,E2 18570.238} C_VEL
LIN {X 0,Y 300.134,Z 702.442,A -85,B 0,C 180,E1 18571.541,E2 18571.541} C_VEL
LIN {X 0,Y 284.984,Z 736.264,A -85,B 0,C 180,E1 18575.172,E2 18575.172} C_VEL
LIN {X 0,Y 267.621,Z 768.453,A -85,B 0,C 180,E1 18580.385,E2 18580.385} C_VEL
LIN {X 0,Y 251.758,Z 794.363,A -85,B 0,C 180,E1 18586.671,E2 18586.671} C_VEL
LIN {X 0,Y 237.797,Z 816.418,A -85,B 0,C 180,E1 18594.614,E2 18594.614} C_VEL
LIN {X 0,Y 227.125,Z 834.176,A -85,B 0,C 180,E1 18604.617,E2 18604.617} C_VEL
LIN {X 0,Y 222.209,Z 844.694,A -85,B 0,C 180,E1 18614.236,E2 18614.236} C_VEL
LIN {X 0,Y 220.918,Z 849.544,A -85,B 0,C 180,E1 18622.146,E2 18622.146} C_VEL
LIN {X 0,Y 220.955,Z 851.178,A -85,B 0,C 180,E1 18629.998,E2 18629.998} C_VEL
LIN {X 0,Y 220.895,Z 849.544,A -85,B 0,C 180,E1 18637.851,E2 18637.851} C_VEL
LIN {X 0,Y 222.805,Z 843.278,A -85,B 0,C 180,E1 18647.392,E2 18647.392} C_VEL
LIN {X 0,Y 228.822,Z 831.103,A -85,B 0,C 180,E1 18657.49,E2 18657.49} C_VEL
LIN {X 0,Y 239.726,Z 813.22,A -85,B 0,C 180,E1 18666.725,E2 18666.725} C_VEL
LIN {X 0,Y 254.742,Z 789.627,A -85,B 0,C 180,E1 18674.703,E2 18674.703} C_VEL
LIN {X 0,Y 271.857,Z 761.086,A -85,B 0,C 180,E1 18680.994,E2 18680.994} C_VEL
LIN {X 0,Y 287.781,Z 730.523,A -85,B 0,C 180,E1 18685.541,E2 18685.541} C_VEL
LIN {X 0,Y 300.233,Z 701.148,A -85,B 0,C 180,E1 18688.695,E2 18688.695} C_VEL
LIN {X 0,Y 296.211,Z 680.591,A -85,B 0,C 180,E1 18694.356,E2 18694.356} C_VEL
LIN {X 0,Y 290.752,Z 662.829,A -85,B 0,C 180,E1 18700.752,E2 18700.752} C_VEL
LIN {X 0,Y 286.07,Z 650.647,A -85,B 0,C 180,E1 18707.048,E2 18707.048} C_VEL
LIN {X 0,Y 282.508,Z 641.181,A -85,B 0,C 180,E1 18715.408,E2 18715.408} C_VEL
LIN {X 0,Y 281.846,Z 639.74,A -85,B 0,C 180,E1 18720.003,E2 18720.003} C_VEL
LIN {X 0,Y 282.304,Z 640.478,A -85,B 0,C 180,E1 18724.602,E2 18724.602} C_VEL
LIN {X 0,Y 284.538,Z 648.832,A -85,B 0,C 180,E1 18732.251,E2 18732.251} C_VEL
LIN {X 0,Y 284.989,Z 649.922,A -85,B 0,C 180,E1 18733.075,E2 18733.075} C_VEL
LIN {X 0,Y 284.862,Z 654.592,A -85,B 0,C 180,E1 18734.587,E2 18734.587} C_VEL
LIN {X 0,Y 284.112,Z 662.963,A -85,B 0,C 180,E1 18736.706,E2 18736.706} C_VEL
LIN {X 0,Y 284.286,Z 663.444,A -85,B 0,C 180,E1 18736.986,E2 18736.986} C_VEL
LIN {X 0,Y 296.142,Z 678.091,A -85,B 0,C 180,E1 18747.3,E2 18747.3} C_VEL
LIN {X 0,Y 304.264,Z 685.638,A -85,B 0,C 180,E1 18753.816,E2 18753.816} C_VEL
LIN {X 0,Y 312.771,Z 693.545,A -85,B 0,C 180,E1 18761.335,E2 18761.335} C_VEL
LIN {X 0,Y 318.327,Z 699.053,A -85,B 0,C 180,E1 18766.928,E2 18766.928} C_VEL
LIN {X 0,Y 322.238,Z 702.126,A -85,B 0,C 180,E1 18770.967,E2 18770.967} C_VEL
LIN {X 0,Y 326.411,Z 706.901,A -85,B 0,C 180,E1 18776.323,E2 18776.323} C_VEL
LIN {X 0,Y 331.629,Z 710.202,A -85,B 0,C 180,E1 18782.935,E2 18782.935} C_VEL
LIN {X 0,Y 334.672,Z 714.257,A -85,B 0,C 180,E1 18788.857,E2 18788.857} C_VEL
LIN {X 0,Y 337.299,Z 716.201,A -85,B 0,C 180,E1 18794.431,E2 18794.431} C_VEL
LIN {X 0,Y 339.333,Z 717.074,A -85,B 0,C 180,E1 18799.755,E2 18799.755} C_VEL
LIN {X 0,Y 340.53,Z 717.489,A -85,B 0,C 180,E1 18804.917,E2 18804.917} C_VEL
LIN {X 0,Y 340.899,Z 717.555,A -85,B 0,C 180,E1 18810.001,E2 18810.001} C_VEL
LIN {X 0,Y 340.501,Z 717.438,A -85,B 0,C 180,E1 18815.086,E2 18815.086} C_VEL
LIN {X 0,Y 338.866,Z 716.965,A -85,B 0,C 180,E1 18821.56,E2 18821.56} C_VEL
LIN {X 0,Y 335.995,Z 715.427,A -85,B 0,C 180,E1 18828.325,E2 18828.325} C_VEL
LIN {X 0,Y 332.768,Z 711.919,A -85,B 0,C 180,E1 18834.909,E2 18834.909} C_VEL
LIN {X 0,Y 329.299,Z 708.626,A -85,B 0,C 180,E1 18840.271,E2 18840.271} C_VEL
LIN {X 0,Y 323.326,Z 703.945,A -85,B 0,C 180,E1 18847.491,E2 18847.491} C_VEL
LIN {X 0,Y 318.313,Z 699.037,A -85,B 0,C 180,E1 18853.075,E2 18853.075} C_VEL
LIN {X 0,Y 311.804,Z 692.388,A -85,B 0,C 180,E1 18859.644,E2 18859.644} C_VEL
LIN {X 0,Y 304.246,Z 685.691,A -85,B 0,C 180,E1 18866.215,E2 18866.215} C_VEL
LIN {X 0,Y 295.186,Z 677.148,A -85,B 0,C 180,E1 18873.426,E2 18873.426} C_VEL
LIN {X 0,Y 282.585,Z 658.986,A -85,B 0,C 180,E1 18885.792,E2 18885.792} C_VEL
